(* CoDeSys 2.3 project: cy-wg-120-001.pro *)
(* Title: cy-wg-24 - ClevergyAS *)
(* Author: Andrea Laini *)
(* Libraries: mod_com.lib 16.5.13 14:00:50, SerComm.lib 16.5.13 14:00:50, Serial_Interface_01.lib 22.4.13 12:50:14, WagoLibLed.lib 17.6.13 10:40:56, Modb_l05.lib 13.5.15 10:30:08, Util.lib 16.5.13 14:00:50, SysLibFile.lib 16.5.13 14:00:50, SysLibRtc.lib 16.5.13 14:00:50, SysLibSockets.lib 22.5.14 16:16:32, SysLibEvent.lib 16.5.13 14:00:50, SysLibPlcCtrl.lib 16.5.13 14:00:50, Standard.lib 20.5.14 08:13:26, Iecsfc.lib 16.5.13 14:00:50, SYSLIBCALLBACK.LIB 16.5.13 14:00:50 *)

(* PLC configuration (modules and I/O channels)
0750-9999/0400-0004 4 DI Generic [Type_1_4_Channels] node 0, in %IB0 out %QB0
  VPN_ST2 AT %IX0.0 [BOOLOnX_I] I 1: Digital Input
  INT01 AT %IX0.1 [BOOLOnX_I] I 2: Digital Input
  KEY_QE_ST AT %IX0.2 [BOOLOnX_I] I 3: Digital Input
  INT02 AT %IX0.3 [BOOLOnX_I] I 4: Digital Input
Modbus variables [PFC200MODBUS] node 1, in %IB0 out %QB0 {PlcStopBehaviour = 1; FiledbusErrorBehaviour = 1; TcpOperation = 0; TcpPort = 502; TcpTimeout = 600; UdpOperation = 0; UdpPort = 502; RtuOperation = 0; NodeId = 200; ResponseTimeout = 5000; Interface = 0; Baud = 38400; StopBits = 2; Parity = 0; FlowCtrl = 0; PhysInterface = 1}
Modbus-Master [MB_MASTER] node 2, in %IB0 out %QB0
*)

(* Task configuration *)
TASK Main (PRIORITY := 6, INTERVAL := T#10ms);
	PLC_PRG();
END_TASK
TASK SystemCheck (PRIORITY := 14, INTERVAL := T#50ms);
	PLC_SYS_FAST();
END_TASK
TASK RTC (PRIORITY := 15, INTERVAL := T#500ms);
	RTC_Update();
END_TASK

(* Global variable list: Global_Constants *)
VAR_GLOBAL CONSTANT

	Plant_NAME			: STRING :='cySN:120 ITB CENE SOLARFAST cyVER:1';
	Plant_SN			: DWORD  :=120;		(* S/N Impianto di telecontrollo *)
	Plant_SW_VER		: WORD   :=1;		(* Versione SW installata *)

	Plant_INV			: BYTE	 :=2;
	Plant_STR			: BYTE	 :=6;

	(* Filesystem *)
	FilesPath  			: STRING :='/media/sd/';

	(* Colour Visu *)
	COLOR_RED			: DWORD := 16#2020F0;
	COLOR_YELLOW		: DWORD	:= 16#20F0F0;
	COLOR_GREEN			: DWORD	:= 16#20F020;

	(* TCP Logger *)
	Logger_SERVER		: STRING:='';
	Logger_IP			: STRING:='178.33.227.41';
	Logger_PORT			: WORD  :=80;
	Logger_GETSTART		: STRING:='GET /cygmsrv/SFgm.ashx?';
	Logger_GETEND		: STRING:='$R$N$R$N';
	Logger_CHECK		: STRING:='True';
	Logger_CRLF			: STRING:='$R$N';
	Logger_DataFile		: STRING:='/media/sd/LOG.DAT';
	Logger_DataFileOld	: STRING:='/media/sd/LOG.BCK';
	Logger_IndexFile	: STRING:='/media/sd/LOG.IDX';
	Logger_ConnRetries	: BYTE:=5;
	Logger_RecoverMsgs	: BYTE:=25;

	(* TCP Remote *)
	Remote_PORT			: WORD  :=10;
	Remote_WELCOME		: STRING:='Connected$R$N';
	Remote_OK			: STRING:='OK$R$N';
	Remote_ERROR		: STRING:='ERROR$R$N';

	(* TCP Sockets *)
	MAX_SEND_TCP_SERVER					 : DWORD:=3000;(*60000*)
	MAX_RECEIVE_TCP_SERVER				 : DWORD:=3000;
	MAX_RECEIVE_TCP_SERVER_SOCKET	 	 : DWORD:=1500;
	MAX_SEND_TCP_CLIENT					 : DWORD:=3000;(*15000*)
	MAX_RECEIVE_TCP_CLIENT				 : DWORD:=1500;
	MAX_RECEIVE_TCP_CLIENT_SOCKET		 : DWORD:=1500;
	MAX_RECEIVE_UDP_SERVER				 : INT  :=1472;
	MAX_RECEIVE_UDP_CLIENT				 : INT  :=1472;
	CONNECT_WATCHDOG_TIME				 : TIME :=t#10s;

END_VAR

(* Global variable list: Global_Retain *)
VAR_GLOBAL RETAIN PERSISTENT
	Mode_Manual : BOOL := FALSE;

	(* Offset correction in case of energy counter reset *)
	Offset		:	ARRAY [1..Plant_INV] OF DINT;

	(* Last value read (Stored in nvm to be sure that in case of a register reset after a voltage dropout, accumulated energy
       is not lost)	*)
	Old_Esup	:	ARRAY [1..Plant_INV] OF DINT;

END_VAR

(* Global variable list: Global_Variables *)
VAR_GLOBAL

	SYS    	: 	typ_SYS;
	Logger 	: 	typ_Logger;

	Lamp	:	LAMP_AL_GENERALE; (* Per gestione allarme generico impianto *)

	(**** PLANT OBJECTS ****)

	(* Define the handler for the ModBus communication	*)
	MODB01		:	obj_MODBUS := (ID:=1, COM:=0, BAUDRATE:=BAUD_38400, RS485:=TRUE);

	(* Define handlers for different objects in the plant; using array permits a better and immediate access *)
	INV			:	ARRAY[1..Plant_INV] OF obj_MODBUS_INV_SUNWAYTG;
	STR			:	ARRAY[1..Plant_STR] OF obj_MODBUS_STR_ES889;

	(**** SIMULATION ONLY ****)
	(*...*)
END_VAR

(* Data type in Logger *)
TYPE en_Logger_ErrLev :
(
	EL_Log			:=0,
	EL_Wrn			:=1,
	EL_Alarm		:=2,
	EL_AlarmStop	:=3,

	EL_Evt			:=4
);
END_TYPE

(* Data type in Logger *)
TYPE en_Logger_Status :
(
	S_Logger_UNKNOWN := 0,
	S_Logger_IDLE,
	S_Logger_WAITCONN,
	S_Logger_WAITTX,
	S_Logger_WAITRESP,
	S_Logger_ERROR
);
END_TYPE

(* Data type *)
TYPE en_SYS_Objects :
(
	EO_SYS		:=0,  (* PLC *)
	EO_VPN		:=1,  (* VPN *)
	EO_DOOR		:=2,  (* Door & access control *)

(*NEW*)EO_SWITCH	:= 3,

	EO_CAL		:=10, (* Caldaia *)
	EO_CIR		:=11, (* Circolatore *)
	EO_CRON		:=12, (* Crono-termostato *)
	EO_VRD		:=13, (* Valvola miscelatore pannelli *)
	EO_CTL		:=14, (* Contalitri *)
	EO_CTB		:=15, (* Contabilizzatore *)
	EO_TPV		:=16, (* Temperature probes values *)
	EO_PPV		:=17, (* Pressure probes values *)
	EO_PBV		:=18, (* Over-Pressure Alarms *)
	EO_TBV		:=19, (* Over-Temperature Alarms *)
	EO_PMV		:=20, (* Under-Pressure Alarms *)
	EO_GRU		:=21, (* Gruppo termico *)
	EO_PDC		:=22, (* Pompa di calore *)
	EO_SOL		:=23, (* Pannello solare termico *)
	EO_ESOL		:=24, (* Pannello solare fotovoltaico *)
	EO_GAS		:=25, (* Contatore GAS *)
	EO_PORT		:=26, (* Misuratore di portata *)
	EO_FPV		:=27, (* Flow probes values *)
	EO_ANZ		:=28, (* Analizzatore di rete *)
	EO_SCA		:=29, (* Signal Control Alarms *)
	EO_LUX		:=30, (* Illumination point *)
	EO_PSG		:=31, (* Sensore di passaggio *)

(*NEW*)EO_INV		:=36, (* Inverter *)
(*NEW*)EO_STR		:=37, (* Smart string box *)

	EO_ZGW			:=200,  (* ZigBee - Gateway *)
	EO_ZRM			:=201,	(* ZigBee - Repeater *)
	EO_ZREL			:=202,	(* ZigBee - Actuator rele *)
	EO_ZTHL			:=203,	(* ZigBee - Temperature Sensor *)

	EO_ASGW			:=250,	(* ASi - Gateway *)
	EO_ASCBI		:=251,	(* ASi - Input Board, Ciabatta *)

	EO_LON			:=1000, (* Bus - LON *)
	EO_MODBUS		:=1001, (* Bus - MODBUS *)
	EO_MBUS			:=1002, (* Bus - M-BUS *)
	EO_MODBUS_TCP	:=1003, (* Bus - MODBUS TCP *)

	EO_GENERIC		:=9000, (* Generic dataset *)
	EO_EXPO			:=9001 (* EXPO dataset *)
);
END_TYPE

(* Data type *)
TYPE en_SYS_Status :
(
	S_UNKNOWN  := 0,
	S_STARTUP,
	S_INIT_RTC,
	S_INIT_VAR,
	S_AUTOTEST,
	S_RUNNING,
	S_SHUTDOWN,
	S_HALT
);
END_TYPE

(* Data type in Logger *)
TYPE typ_Logger :
STRUCT
	Status		: en_Logger_Status;

	SendReq		: BOOL;
	SendIdx		: DWORD;
	SendData	: ARRAY [0..MAX_SEND_TCP_CLIENT] OF BYTE;
	SendLen		: DINT;

	TData		: ARRAY [0..MAX_SEND_TCP_CLIENT] OF BYTE;
	TLen		: DINT;

	LastIdxPos	: DWORD;

	(* Temporary variables used by objects *)
	s1			: STRING(256);
	i1			: WORD;

END_STRUCT
END_TYPE

(* Data type in Plant_Objects *)
TYPE typ_MODBUS_INV_SUNWAYTG : (* updated by Diego Bernini on 2016-02-18 *)
STRUCT
		(**** General measurements (see Programming manual) ****)
		Vpv_ref		:	WORD;	(* e-1 V*)
		f			:	INT;	(* e-2 Hz *)
		pf			:	WORD;	(* e-2 *)
		P			:	INT;	(* e-1 kW *)	(* Power supplied to the net b the inverter *)
		Pr			:	INT;	(* e-1 kVAr *)	(* Reactive power supplied to the net b the inverter *)
		Pa			:	INT;	(* e-1 kVA *)	(* Appearent power supplied to the net b the inverter *)
		Vinv		:	WORD;	(* e-1 V *)		(* Inverter output voltage, before output tf *)
		Vmain	 	:	WORD;	(* e-1 V *)		(* Main voltage, after output tf *)
		Iinv		:	WORD;	(* e-1 A *)		(* As voltage *)
		Imain		:	WORD;	(* e-1 A *)		(* AS voltage *)
		Vpv			:	WORD;	(* e-1 V *)		(* PV field voltage measured by the inverter *)
		Ipv			:	WORD;	(* e-1 A *)		(* PV current measured by the inverter *)
		Ppv			:	INT;	(* e-1 kW *)	(* Power generated by the PV *)

		(**** Energy ****)
		Esup_ExtCtr1:	DINT;	(* e-2 kWh *)	(* Global active energy supplied to the net *) (* updated *)
		ExtCtr2		:	DINT;	(* e-2 kWh *)
		Epv			:	DWORD;	(* e-2 kWh *)	(* Global produced energy since start *)

		(**** Temeprature ****)
		Tboard		:	INT;	(* e-1 °C *)	(* Control board temperature *)
		Tigbt		:	INT;	(* e-1 °C *)	(* Igbt temperature *)

		(**** Digital Input ****)
		ClampStatus	:	WORD;

		(**** Main measurements (otherwise not specified, all measurements are referred to the mains, therefore AFTER output tf ****)
		Vrms_rs		:	WORD;	(* e-1 V *)
		Vrms_st		:	WORD;
		Vrms_tr		:	WORD;
		Irms_r		:	INT;	(* e-1 A *)
		Irms_s		:	INT;
		Irms_t		:	INT;
		PLLStatus	:	WORD;
		MainStatus2	:	WORD;
		MainStatus1	:	WORD;
		Iinv_rms_r	:	INT;	(* e-1 A *)		(* Measured between inverter and tf *)
		Iinv_rms_s	:	INT;
		Iinv_rms_t	:	INT;
		Iimbalance	:	WORD;	(* e-1 *)
		Vrms_r		:	WORD;	(* e-1 V *)
		Vrms_s		:	WORD;
		Vrms_t		:	WORD;
		P_r			:	INT;	(* e-1 kW *)
		P_s			:	INT;
		P_t			:	INT;
		Pr_r		:	INT;	(* e-1 kW *)
		Pr_s		:	INT;
		Pr_t		:	INT;

		(**** Inverter Status (see Programming manual) ****)
		Status		:	WORD;
		ActiveAlarm	:	WORD;
		Insulation	:	WORD;
		Event		:	WORD;
		OpTime		:	DWORD;	(* e-0.7 s *)
		SuppTime	:	DWORD;	(* e-0.7 s *)

END_STRUCT
END_TYPE

(* Data type in Plant_Objects *)
TYPE typ_MODBUS_INV_SUNWAYTG_His :
STRUCT
		AlarmID		:	WORD;
		SuppTime	: 	DWORD;
		OpTime		:	DWORD;
		InvStatus	:	WORD;
		Vpv_ref		:	WORD;
		Vpv			:	WORD;
		Vmain		:	WORD;
		Status2		:	WORD;
		Status1		:	WORD;
		Tboard		:	INT;
		Tigbt		:	INT;
		I_u			:	INT;
		I_v			:	INT;
		I_w			:	INT;
		ClampStatus	:	WORD;
		DigOutput	:	WORD;
		IgbtFault	:	WORD;
		Psupp		:	DWORD;
		Epv			:	DWORD;

END_STRUCT
END_TYPE

(* Data type in Plant_Objects *)
TYPE typ_MODBUS_STR_ES889 :
STRUCT

	(* GENERAL MEASUREMENTS *)
	(* String current *)
	Istring1	:	WORD;			(* e-2 A *)
	Istring2	:	WORD;
	Istring3	:	WORD;
	Istring4	:	WORD;
	Istring5	:	WORD;
	Istring6	:	WORD;
	Istring7	:	WORD;
	Istring8	:	WORD;
	Iavg		:	WORD;
	Imax		:	WORD;
	Imin		:	WORD;

	(* Optional sensors *)
	Radiation_h	:	WORD;			(* e-1 W/m2	,	Radiation on the horizontal plane *)
	Radiation_m	:	WORD;			(*			,	Radiation on modules plane *)
	Tmodule		:	INT;			(* e-1 °C	,	Module temperature *)
	Tenv		:	INT;			(*			,	Environment temperature *)
	Vwind		:	WORD;			(* e-1 m/s	,	Wind speed *)
	Tboard		:	INT;			(* e-1 °C	,	Board temperature *)

	(* FUNCTIONING STATUS *)
	M018		:	WORD;
	M019		:	WORD;
	M020		:	WORD;

	(* TIMING *)
	SuppTime	:	DWORD;			(* s ???? *)
	OpTime		:	DWORD;			(* s ???? *)

	(* String mask	*)
	Mask		:	WORD;

	(* Panels number	*)
	Panels		:	WORD;

END_STRUCT
END_TYPE

(* Data type in Plant_Objects *)
TYPE typ_MODBUS_STR_ES889_His :
STRUCT

	M018		:	WORD;
	M020		:	WORD;
	Tmodule		:	INT;			(* e-1 °C	,	Module temperature *)
	SuppTime	:	DWORD;
	OpTime		:	DWORD;

END_STRUCT
END_TYPE

(* Data type in Plant_Objects *)
TYPE typ_MODBUS_VAR : (* Gestione parametri MODBUS *)
STRUCT
	SlaveAddress	: BYTE;
	FunCode			: BYTE;
	FunAddress		: WORD;
	Refresh_Time	: BYTE; (* 0:No refresh x:Refresh in seconds *)
	Refresh_Cnt		: BYTE; (* INTERNAL *)
	Variable		: POINTER TO ARRAY [0..124] OF WORD;	(* For classical ModBus it has to be equal to "typModbusResponse.Data"
																that is an array of 125 word ([0..124]) *)
	Variable_Size	: BYTE;
	Variable_Mirror : WORD; (* INTERNAL [Force refresh on read variables when <>0] *)
END_STRUCT
END_TYPE

(* Data type *)
TYPE typ_SYS :
STRUCT
	Status			: en_SYS_Status;
	Warning			: BOOL;
	Alarm			: BOOL;
	AlarmStop		: BOOL;

	Time_LogString	: STRING;
	Time_Year		: WORD;
	Time_Month		: BYTE;
	Time_Day		: BYTE;

	Time_CT_DT		: DT;
	Time_CT_Day		: WORD;
	Time_CT_Quarter	: BYTE;

	LastLogs_Idx	: BYTE;
	LastLogs_Dat	: ARRAY[0..5] OF STRING;
	LastLogs_Msg	: ARRAY[0..5] OF STRING;

END_STRUCT
END_TYPE

(* Data type in Plant_Objects *)
TYPE typ_VisuStrutturaMbus :
STRUCT

	sdNodoPresente: STRING(16);
	sdEnergia: STRING(16);
	sdPotenza: STRING(16);
	sdVolume: STRING(16);
	sdFlow: STRING(16);
	sdTempIngresso: STRING(8);
	sdTempaUscita: STRING(8);
	sdTempDelta: STRING(8);

END_STRUCT
END_TYPE

(* POU PLC_PRG, ST *)
PROGRAM PLC_PRG
VAR
	Timer1: TON; (* Logger timer *)

	i	  : BYTE;
	status : BYTE;
END_VAR
(******************************************************************************
 ****        		MAIN TASK CODE  (called every 10ms)                    ****
 ******************************************************************************

	Network setup:
		IP  = 192.168.100.2 | MSK = 255.255.255.0
		GW	= 192.168.100.1 | DNS = 192.168.100.1
		SNTP = 193.204.114.232 (3600s) ==> 192.168.100.3

*)

(*==============================*)
(*===== Main status machine ====*)
(*==============================*)
Main_Stm();

(*==============================*)
(*== Running cycle operations ==*)
(*==============================*)
IF SYS.Status>S_INIT_VAR THEN
	(* Execute cycle processes *)
	MODB01();

	FOR i:=1 TO Plant_INV BY 1 DO INV[i](ModBus:=MODB01, retryErrMax:=1);	END_FOR

	FOR i:=1 TO Plant_STR BY 1 DO STR[i](ModBus:=MODB01, retryErrMax:=1);   END_FOR

END_IF

(*==============================*)
(*== System cycle operations ===*)
(*==============================*)
(* Execute TCP processes *)
Logger_Proc();
Remote_Proc();
(* Update user led *)
(*USRLED_Update();*)
(* Execute Cron Editor commands *)
(*
CronEd();
*)
(* External resources *)
(*

*)

(**** SIMULATION ONLY ****)
(*...*)
END_PROGRAM
ACTION Main_Stm:
CASE Sys.Status OF

	S_STARTUP:
		Sys.Status:=S_INIT_RTC;

	S_INIT_RTC:
		(* Check RTC and update from network *)
		RTC_Update();
		(* Check time *)
		IF Sys.Time_Year>2000 THEN
			Sys.Status:=S_INIT_VAR;
		END_IF

	S_INIT_VAR:
		OBJ_Definition();

		LogEv(EL_Wrn,EO_SYS,0,1,CONCAT('System_startup_v',WORD_TO_STRING(Plant_SW_VER)));
		Sys.Status:=S_RUNNING;

	S_RUNNING:

		status :=0;
		FOR i:=1 TO Plant_INV BY 1 DO IF INV[i].Status_Log=1 THEN status :=1;  END_IF	END_FOR

		FOR i:=1 TO Plant_STR BY 1 DO IF str[i].Status_Log=1 THEN status :=1; END_IF END_FOR

		FOR i:=1 TO Plant_INV BY 1 DO IF INV[i].Status_Log=2 THEN status :=2;  END_IF	END_FOR

		FOR i:=1 TO Plant_STR BY 1 DO IF str[i].Status_Log=2 THEN status :=2; END_IF END_FOR

		Lamp( Allarme:=	(status=2),
			  Warning:=  (status=1),
			  SistemaInAllarme => Sys.Alarm,
			 SistemaWarning => Sys.Warning
			 );

		Timer1(IN:=NOT Timer1.Q,PT:=T#5m);
		IF Timer1.Q THEN
			(* Trig logger *)
			LogTrig();
			(* Execute temporary CSV logger *)
			(*CSV_Log();*)
		END_IF

	S_SHUTDOWN:
		(* Stop sistema *)
		Sys.Status:=S_STARTUP;

	S_HALT:
		(* Aspetta uscita manuale *)
		Sys.Status:=S_STARTUP;

ELSE
	Sys.Status:=S_STARTUP;
END_CASE;
END_ACTION
ACTION OBJ_Definition:
(**** Define Plant Objects ****)

(* Inverter *)
INV[1].ID := 1;		INV[1].Address := 2;
INV[2].ID := 2;		INV[2].Address := 3;


(* StringBox *)
STR[1].ID := 1;		    STR[1].Address :=10;
STR[2].ID := 2;		    STR[2].Address := 11;
STR[3].ID := 3;		    STR[3].Address := 12;
STR[4].ID := 4;		    STR[4].Address := 13;
STR[5].ID := 5;		    STR[5].Address := 14;
STR[6].ID := 6;		    STR[6].Address := 15;
END_ACTION

(* POU TCP_Logger/Logger_Proc, ST *)
PROGRAM Logger_Proc
VAR
	c1:         	TCPCLIENT;

	Open:	    	BOOL;
	IpAddr:			DWORD;
	InetAddr:		DWORD;
	Connected:  	BOOL;
	Error:      	DINT;
	TxTrig:     	BOOL;
	RxData:			ARRAY [0..MAX_RECEIVE_TCP_CLIENT] OF BYTE;
	RxLen:			DINT;

	Retry:			BYTE;	(* Counter for connection retries *)
	Recovered:		BYTE;	(* Counter for recovered unsent messages *)

	i:				DINT;
	pos:			DWORD;
	hFile:			DWORD;

END_VAR
(*=== State machine ===*)
CASE Logger.Status OF

	S_Logger_UNKNOWN:
		(* Startup *)
		Logger.SendReq:=FALSE;
		Open:=FALSE;
		Logger.Status:=S_Logger_IDLE;

	S_Logger_IDLE:
		(* Wait request *)
		IF Logger.SendReq THEN
			(* Resolve server name or use static IP *)
			IF LEN(Logger_SERVER)=0 THEN
				InetAddr:=SysSockInetAddr(Logger_IP);
			ELSE
				IpAddr:=SysSockGetHostByName(ADR(Logger_SERVER));	(* Get the IP address by the DNS *)
				DWORDSWAP(pIn:=ADR(IpAddr), pOut:=ADR(InetAddr));
			END_IF
			TxTrig:=FALSE;
			RxLen:=0;
			(* Open connection *)
			Open:=TRUE;
			Logger.Status:=S_Logger_WAITCONN;
		END_IF

	S_Logger_WAITCONN:
		(* Wait connection *)
		IF Connected THEN
			(* Send data *)
			TxTrig:=TRUE;
			Logger.Status:=S_Logger_WAITTX;
		END_IF
		IF Error>0 THEN
			Open:=FALSE;
			Logger.Status:=S_Logger_ERROR;
		END_IF

	S_Logger_WAITTX:
		(* Wait transmission *)
		IF NOT TxTrig THEN
			Logger.Status:=S_Logger_WAITRESP;
		END_IF
		IF Error>0 THEN
			Open:=FALSE;
			Logger.Status:=S_Logger_ERROR;
		END_IF

	S_Logger_WAITRESP:
		(* Wait response *)
		IF Connected=FALSE (* OR TIMEOUT!! *) THEN
			Open:=FALSE;
			(* Check response *)
			IF RxLen>=4 AND CHKSTRING(pString:=ADR(RxData), pPattern:=ADR(Logger_CHECK)) THEN
			(* If "RxLen" is of the right size and function "CHKSTRING" has not return "FALSE"	*)
				Logger.SendReq:=FALSE;
				Retry:=0;
				(* Check unsent messages to flush *)
				IF Recovered<Logger_RecoverMsgs THEN
					MsgChk();
					IF Logger.SendReq=TRUE THEN
						Recovered:=Recovered+1;
					ELSE
						Recovered:=0;
					END_IF
				ELSE
					Recovered:=0;
				END_IF
				Logger.Status:=S_Logger_IDLE;
			ELSE
				Logger.Status:=S_Logger_ERROR;
			END_IF
		END_IF

	S_Logger_ERROR:
		(* Connection error or send failure *)
		Retry:=Retry+1;
		IF Retry>Logger_ConnRetries THEN
			(* Save message as unsent *)
			MsgSave();
			Logger.SendReq:=FALSE;
			Retry:=0;
		END_IF
		Logger.Status:=S_Logger_IDLE;

ELSE
	Logger.Status:=S_Logger_UNKNOWN;
END_CASE


(*=== Execute client lib ===*)
c1(
	xOpenConnection			:= Open,
	dwInetAddr 				:= InetAddr,
	wPortNumber				:= Logger_PORT,
	ptSendData				:= ADR(Logger.SendData),
	diSendCount				:= Logger.SendLen,
	tConnectWatchdogTime	:= t#10s,
	xStartSend				:= TxTrig,
	aReceiveBuffer			:= RxData,
	diReceiveCount			:= RxLen,
	xConnected				=> Connected,
	diError					=> Error
);

(*=== Process Rx data ===*)
(*IF RxLen>0 THEN
	RxLen:=0;
END_IF*)
END_PROGRAM
ACTION MsgChk:
(* Open index file *)
hFile:=SysFileOpen(Logger_IndexFile,'r');
IF hFile=0 THEN
	(* File doesn't exist, no pending message *)
	RETURN;
END_IF
(* Search oldest message to recover *)
SysFileSetPos(hFile,Logger.LastIdxPos);		(* Set the pointer to last position *)
Logger.SendLen:=0;
REPEAT
	SysFileRead(hFile, ADR(Logger.SendIdx), SIZEOF(Logger.SendIdx));
	pos:=SysFileGetPos(hFile);
	SysFileRead(hFile, ADR(Logger.SendLen), SIZEOF(Logger.SendLen));
UNTIL
	SysFileEOF(hFile) OR Logger.SendLen<>0		(* If equal to 0 means data not stored or deleted *)
END_REPEAT
SysFileClose(hFile);
(* Delete index file when all messages are recovered *)
IF Logger.SendLen=0 THEN
	Logger.LastIdxPos:=0;
	SysFileDelete(Logger_IndexFile);
	RETURN;
END_IF
(* Recover message data *)
hFile:=SysFileOpen(Logger_DataFile,'r');
IF hFile<>0 THEN
	SysFileSetPos(hFile,Logger.SendIdx);
	SysFileRead(hFile,ADR(Logger.SendData),Logger.SendLen);
	Logger.SendReq:=TRUE;									(* Re-trigger another transmission *)
	SysFileClose(hFile);
END_IF
(* Clear index entry *)
hFile:=SysFileOpen(Logger_IndexFile,'a');
IF hFile<>0 THEN
	SysFileSetPos(hFile,pos);
	i:=0;
	SysFileWrite(hFile, ADR(i), 4);			(* Since the size is in number of byte, that clears only the Idx, not the Len *)
	Logger.LastIdxPos:=SysFileGetPos(hFile);
	SysFileClose(hFile);
END_IF
END_ACTION
ACTION MsgSave:
(* Add log position in recovery indexes *)
hFile:=SysFileOpen(Logger_IndexFile,'a');
SysFileWrite(hFile, ADR(Logger.SendIdx), SIZEOF(Logger.SendIdx));
SysFileWrite(hFile, ADR(Logger.SendLen), SIZEOF(Logger.SendLen));
SysFileClose(hFile);
END_ACTION

(* POU Utils Functions/TCPCLIENT, ST *)
FUNCTION_BLOCK TCPCLIENT
(***********************************************************************************************************	*)
(* Version: 1.3b                        			          													*)
(* Date: 28.10.2014                   				          							            			*)
(***********************************************************************************************************	*)
(* WAGO Kontakttechnik GmbH Hansastr. 27 32423 Minden(Westf.)													*)
(* Tel. +0049 571/887-0 Fax. +0049 571/887-0																	*)
(* Author: VB																									*)
(***********************************************************************************************************	*)
(*Description:	A TCP client to read and write data with additional connection watchdog							*)
(*History:																										*)
(*Version 1.3b: 28.10.2014: Use DWORD address for IP (Andrea Ravasio)											*)
(*Version 1.3: 11.02.2011: Changes according to 750-880/881											 			*)
(*Version 1.2: 29.08.2007 Bugfix TCP Client																		*)
(*Version 1.1: 15.01.2007 Changes according to FW11																*)
(*Version 1.0: 09.03.2006 Release																				*)
(***********************************************************************************************************	*)
VAR CONSTANT
	STATE_CREATE     				 : BYTE:= 0;
	STATE_OPEN     					 : BYTE:= 1;
	STATE_IOCTL    					 : BYTE:= 2;
	STATE_CONNECT     				 : BYTE:= 10;
	STATE_TX       					 : BYTE:= 20;
	STATE_RX       					 : BYTE:= 30;
	STATE_CLOSE    					 : BYTE:= 40;
	STATE_ERROR_TRAP			     : BYTE:= 200;
END_VAR

VAR_INPUT
	xOpenConnection					: BOOL;
	dwInetAddr						: DWORD; (* <== Use SysSockInetAddr() value or
													swapped bytes order of SysSockGetHostByName() value *)
	wPortNumber						: WORD;
	ptSendData						: POINTER TO ARRAY[0..MAX_SEND_TCP_CLIENT] OF BYTE;
	diSendCount						: DINT;
	tConnectWatchdogTime		    : TIME := t#10s;
END_VAR
VAR_OUTPUT
	xConnected						: BOOL;
	diError 						: DINT := 0;
END_VAR
(* ErrorCodes -----------------------------------------
	16#8001 => No socket descriptor available 
	16#8002 => SysSockSend returns -1 
	16#8003 => Socket was "gracefully closed" 
	16#8004 => switching to none blocking mode fails
	16#8005 => SysSockClose() returns FALSE 
    16#8006 => SysSockConnect() fails
    16#8007 => SysSockSend() fails
	16#8008 => error state machine 
	16#8009 => timeout while waiting for data from server 
------------------------------------------------------------*)
VAR_IN_OUT
	xStartSend							: BOOL;
	aReceiveBuffer						: ARRAY [0..MAX_RECEIVE_TCP_CLIENT] OF BYTE;
	diReceiveCount						: DINT;
END_VAR
VAR
	m_State								: BYTE := 0;
	m_ReceiveBuffer						: ARRAY [0..MAX_RECEIVE_TCP_CLIENT_SOCKET] OF BYTE;
	m_Socket							: DINT;
	m_AddressInfo						: SOCKADDRESS;
	m_BytesReceived						: DINT;
	m_diReturn							: DINT;
	m_xReturn							: BOOL;
	m_IoCtlParameter  					: DINT := 1; (* IOCTL-Parameter for non-blocking mode of sockets *)
	i									: INT;
	T_Connect							: TON;
	m_count								: DINT;
	diOption							: DINT := 1;
	m_Blocking   						: DINT := 0;
END_VAR
IF xOpenConnection THEN
	(* State maschine *)
	CASE  m_State OF

	(* -------------------------------------------------------------------------*)
	STATE_CREATE:
			(* create socket descriptor*)
			m_Socket := SysSockCreate(diAddressFamily	:= SOCKET_AF_INET,
													 diType		:= SOCKET_STREAM,
													 diProtocol := SOCKET_IPPROTO_TCP);
			IF m_Socket >= 0 THEN
			(*Set Push-Bit*)
				IF ADR(%MW0)=16#30000000  OR ADR(%MW0)=16#20000000 THEN (*841 or 881*)
					SysSockSetOption(
						diSocket:=m_Socket,
						diLevel:=6,
						diOption:=SOCKET_TCP_NODELAY,
						pOptionValue:=ADR(diOption),
						diOptionLength:=SIZEOF(diOption));
				ELSE
						;
				END_IF
				m_State := STATE_IOCTL; (* succesful *)
			ELSE
				diError := 16#8001;  (* no socket descriptor available *)
				m_State := STATE_ERROR_TRAP;
			END_IF

	(* -------------------------------------------------------------------------*)
	STATE_IOCTL: (* change  socket mode  to none blocking *)
		m_diReturn := SysSockIoctl( m_Socket, SOCKET_FIONBIO, ADR(m_IoCtlParameter));
		IF m_diReturn <> 0 THEN
			m_AddressInfo.sin_family := SOCKET_AF_INET;
			m_AddressInfo.sin_port := SysSockNtohs(wPortNumber);
			m_AddressInfo.sin_addr := dwInetAddr;
			m_State := STATE_CONNECT;
		ELSE
			diError := 16#8004;  (* switching to none blocking mode fails *)
			m_State := STATE_ERROR_TRAP;
		END_IF


	(* -------------------------------------------------------------------------*)
	STATE_CONNECT: (* connect with server *)
		T_Connect(IN:=TRUE , PT:=tConnectWatchdogTime);(*activate watchdog for establishing connection to a server*)
		m_xReturn := SysSockConnect ( m_Socket, ADR(m_AddressInfo),  SIZEOF(m_AddressInfo));
		IF m_xReturn THEN (* succesful *)
			IF xStartSend THEN
				m_State := STATE_TX;(*transmit data*)
			ELSE
				m_State := STATE_RX;(*wait for data from server*)
			END_IF
			xConnected:=TRUE;
			T_Connect(IN:=FALSE);
		ELSE
			IF T_Connect.Q THEN
				diError := 16#8006;  (* connect fails *)
				xConnected:=FALSE;
				T_Connect(IN:=FALSE);
				m_State := STATE_ERROR_TRAP;
				SysSockClose( m_Socket);
			ELSE
				m_State := STATE_CONNECT;(*client still  tries to set up connection*)
			END_IF
		END_IF


	STATE_TX:	 (* send TCP-message *)
		m_diReturn := SysSockSend(diSocket := m_Socket,
								  pbyBuffer := ADR(ptSendData^[0]),
								  diBufferSize := diSendCount-m_count,
								  diFlags := 0);

		CASE m_diReturn OF
		-1:	(* ERROR *)
			T_Connect(IN:=TRUE , PT:=CONNECT_WATCHDOG_TIME);(*activate watchdog to check communication*)
			IF t_Connect.Q THEN
				diError := 16#8007;
				T_Connect(IN:=FALSE);
				m_State:=STATE_CLOSE;
			END_IF
		0: (* socket was "gracefully closed" *)
			m_State := STATE_CLOSE;
			diError := 16#8003;
		ELSE (* succesful *)
			m_count:=m_count+m_diReturn;
			IF m_count>=diSendCount THEN
				diError := 16#0000;
				m_State := STATE_RX;
				m_count:=0;
				xStartSend:=FALSE;
			END_IF
			T_Connect(IN:=FALSE);
		END_CASE

	(* -------------------------------------------------------------------------*)
	STATE_RX: (* process receive data *)
			m_BytesReceived := SysSockRecv(	diSocket 	:= m_Socket,
										pbyBuffer 	:= ADR(m_ReceiveBuffer),		(* Address of receive buffer *)
										diBufferSize:= SIZEOF(m_ReceiveBuffer),
										diFlags		:= 0);

			CASE m_BytesReceived OF
			-1:	(* No data available or error occured *)
				T_Connect(IN:=TRUE , PT:=tConnectWatchdogTime);(*activate watchdog to check communication*)
				IF t_Connect.Q THEN
					diError:=16#8009;
					T_Connect(IN:=FALSE);
					m_State:=STATE_CLOSE;
				END_IF
				IF xStartSend THEN
					m_State:=STATE_TX	;(* WAIT IN THIS STATE  and check for arriving data or new send command*)
				END_IF;
			0: (* socket was "gracefully closed"  *)
				m_State:=STATE_CLOSE;
				diError := 16#8003;
			ELSE (* succesful *)
				diError := 16#0000;
				T_Connect(IN:=FALSE);
				(* Copy received data into receive buffer *)
				FOR i:= 0 TO DINT_TO_INT(m_BytesReceived	)-1 DO
					aReceiveBuffer[diReceiveCount]:= m_ReceiveBuffer[i];
					diReceiveCount:=(diReceiveCount+1) MOD SIZEOF(aReceiveBuffer);
				END_FOR

			END_CASE

	(* -------------------------------------------------------------------------*)
	STATE_CLOSE : (* close socket *)
		IF ADR(%MW0)=16#30000000  OR ADR(%MW0)=16#20000000 THEN (*841 or 881*)
			;
		ELSE
			SysSockShutdown(m_Socket, 0);;(*870*)
		END_IF
		m_xReturn := SysSockClose( m_Socket);
		m_Socket := -1;
		m_State := 0; (* succesful *)
		xConnected:=FALSE;
		T_Connect(IN:=FALSE);
	(* -------------------------------------------------------------------------*)
	STATE_ERROR_TRAP: (* error handling *)
		xConnected:=FALSE;

	ELSE  (* Bad FSM code trap  *)
			m_State:= STATE_ERROR_TRAP;
			diError:= 16#8008;
	END_CASE

ELSE(*close connection*)
	IF m_Socket >= 0 THEN
		IF ADR(%MW0)=16#30000000  OR ADR(%MW0)=16#20000000 THEN (*841 or 881*)
			;
		ELSE
			SysSockShutdown(m_Socket, 0);;(*870*)
		END_IF
		SysSockClose( m_Socket);
	END_IF
	m_Socket := -1;
	diError := 16#0000;
	m_State := STATE_CREATE;
	xConnected:=FALSE;
	T_Connect(IN:=FALSE);
END_IF
END_FUNCTION_BLOCK

(* POU Utils Functions/DWORDSWAP, ST *)
FUNCTION DWORDSWAP:BOOL
VAR_INPUT
	pIn:POINTER TO ARRAY[1..4] OF BYTE;
	pOut:POINTER TO ARRAY[1..4] OF BYTE;
END_VAR
VAR
END_VAR
pOut^[1]:=pIn^[4];
pOut^[2]:=pIn^[3];
pOut^[3]:=pIn^[2];
pOut^[4]:=pIn^[1];
END_FUNCTION

(* POU Utils Functions/CHKSTRING, ST *)
FUNCTION CHKSTRING : BOOL
VAR_INPUT
	pString: POINTER TO BYTE;
	pPattern: POINTER TO BYTE;
END_VAR
VAR
END_VAR
CHKSTRING:=TRUE;
WHILE pPattern^<>0 AND CHKSTRING DO
	IF pPattern^<>pString^ THEN CHKSTRING:=FALSE; END_IF
	pString:=pString+1;
	pPattern:=pPattern+1;
END_WHILE
END_FUNCTION

(* POU TCP_Remote/Remote_Proc, ST *)
PROGRAM Remote_Proc
VAR
	s1:         	TCPSERVER;
	Enable: 		BOOL;
	Connected: 		BOOL;
	Error: 			DINT;

	TxData:			ARRAY [0..MAX_SEND_TCP_SERVER] OF BYTE;
	TxLen:			DINT;
	TxTrig:			BOOL;

	RxData:			ARRAY [0..MAX_RECEIVE_TCP_SERVER] OF BYTE;
	RxLen:			DINT;

	Status:			DINT;

	(* Command interpreter *)

	Cmd_Buf:		ARRAY [0..MAX_RECEIVE_TCP_SERVER] OF BYTE;
	Cmd_Buf_U16:	POINTER TO WORD;
	Cmd_Buf_INT:	POINTER TO INT;
	Cmd_BufLen:		WORD;
	Cmd_St:			WORD;

	Cmd_Obj:		WORD;
	Cmd_ObjIdx:		WORD;
	Cmd_C:			WORD;
	Cmd_R:			WORD;
	Cmd_CLen:		WORD;
	Cmd_RLen:		WORD;

	i : WORD;
	j : INT;
	s2 : STRING;

	(* per aggiornare la data e l'ora *)
	SetAnno: INT;
	SetMese: INT;
	SetGiorno: INT;
	SetOra: INT;
	SetMinuti: INT;
	SetSecondi: INT;

	Plant_SW_VER: BOOL;
END_VAR
(*=== State machine ===*)
CASE Status OF
	0: (* Startup *)
		TxLen:=0; TxTrig:=FALSE;
		RxLen:=0;
		Enable:=TRUE;
		Status:=1;

	1: (* Wait incoming connection *)
		IF Connected THEN
			(* Log access *)(*
			LogEv(EL_Log,EO_VPN,1,5,'Remote');*)
			(* Send welcome message *)(*
			ADDSTRING(pTxData:=ADR(TxData), pString:=ADR(Remote_WELCOME), TxLen:=TxLen);
			TxTrig:=TRUE;*)
			(* Reset vars *)
			Cmd_BufLen:=0;
			Cmd_St:=0;
			Status:=2;
		END_IF
		IF Error>1 THEN
			Enable:=FALSE;
			Status:=0;
		END_IF

	2: (* Wait command *)
		IF RxLen>0 THEN
			(*=== Interpreter start ===*)
			IF Cmd_BufLen+(RxLen/2)>=MAX_RECEIVE_TCP_SERVER THEN
				(* ERROR *)
				Cmd_BufLen:=0;
			ELSE
				i:=HEXTORAW(pString:=ADR(RxData), StringLen:=DINT_TO_WORD(RxLen), pData:=ADR(Cmd_Buf[Cmd_BufLen]));
				Cmd_BufLen:=Cmd_BufLen+i;
			END_IF
			IF Cmd_BufLen>=8 THEN
				Cmd_Buf_U16:=ADR(Cmd_Buf[6]);
				IF Cmd_BufLen>=(8+Cmd_Buf_U16^) THEN	(* Right number of bytes has been received (8 of protocol + data) *)
					Cmd_CLen:=Cmd_Buf_U16^;
					Cmd_Buf_U16:=ADR(Cmd_Buf[0]); Cmd_Obj:=Cmd_Buf_U16^;
					Cmd_Buf_U16:=ADR(Cmd_Buf[2]); Cmd_ObjIdx:=Cmd_Buf_U16^;
					Cmd_Buf_U16:=ADR(Cmd_Buf[4]); Cmd_C:=Cmd_Buf_U16^;
					(* Log command *)(*
					s2:='RCmd_';		s2:=CONCAT(s2,WORD_TO_STRING(Cmd_Obj));
					s2:=CONCAT(s2,'_'); s2:=CONCAT(s2,WORD_TO_STRING(Cmd_ObjIdx));
					s2:=CONCAT(s2,'_'); s2:=CONCAT(s2,WORD_TO_STRING(Cmd_C));
					s2:=CONCAT(s2,'_');	s2:=CONCAT(s2,WORD_TO_STRING(Cmd_CLen));
					LogEv(EL_Log,EO_VPN,1,6,s2);*)
					(* Execute command *)
					Command();
					Cmd_BufLen:=0;
				END_IF
			END_IF
			(*=== Interpreter end ===*)
			RxLen:=0;
		END_IF
		IF NOT Connected THEN
			Status:=0;
		END_IF

ELSE
	Status:=0;
END_CASE


(*=== Execute server lib ===*)
s1(
	xEnable				:= Enable,
	wPortNumber			:= Remote_PORT,
	tServerTimeOut		:= t#15m,
	ptSendData			:= ADR(TxData),
	diSendCount			:= TxLen,
	xStartSend			:= TxTrig,
	aReceiveBuffer		:= RxData,
	diReceiveCount		:= RxLen,
	xClientConnected	=> Connected,
	diError				=> Error
);
END_PROGRAM
ACTION Cmd_CRON:
(* Check index *)(*
IF Cmd_ObjIdx<1 OR Cmd_ObjIdx>6 THEN
	Cmd_R:=2;
	RETURN;
END_IF

(* Process command *)
CASE Cmd_C OF

	1: (* GET PROFILE *)
		IF Cmd_CLen<>3 THEN
			Cmd_R:=4;
		ELSE
			(* Load profile *)
			CronEd.CN_Sel:=WORD_TO_BYTE(Cmd_ObjIdx);
			Cmd_Buf_U16:=ADR(Cmd_Buf[8]);
			CronEd.CN_YSel:=Cmd_Buf_U16^;
			CronEd.PR_Sel:=Cmd_Buf[10];
			CronEd.PR_Load_Exe();
			(* Copy data *)
			Cmd_RLen:=192;
			TxLen:=TxLen+RAWTOHEX(ADR(CronEd.PR.Setpoint),192,ADR(TxData[TxLen]));
		END_IF

	2: (* SET PROFILE *)
		IF Cmd_CLen<>(3+192) THEN
			Cmd_R:=4;
		ELSE
			(* Save profile *)
			CronEd.CN_Sel:=WORD_TO_BYTE(Cmd_ObjIdx);
			Cmd_Buf_U16:=ADR(Cmd_Buf[8]);
			CronEd.CN_YSel:=Cmd_Buf_U16^;
			CronEd.PR_Sel:=Cmd_Buf[10];
			MEMCPY(ADR(Cmd_Buf[11]),ADR(CronEd.PR.Setpoint),192);
			CronEd.PR_Save_Exe();
		END_IF

	5: (* GET CALENDAR MONTH *)
		IF Cmd_CLen<>3 THEN
			Cmd_R:=4;
		ELSE
			(* Load calendar *)
			CronEd.CN_Sel:=WORD_TO_BYTE(Cmd_ObjIdx);
			Cmd_Buf_U16:=ADR(Cmd_Buf[8]);
			CronEd.CN_YSel:=Cmd_Buf_U16^;
			CronEd.CA_Sel:=Cmd_Buf[10];
			CronEd.CA_Load_Exe();
			(* Copy data *)
			Cmd_RLen:=32;
			TxLen:=TxLen+RAWTOHEX(ADR(CronEd.CA.Profile),32,ADR(TxData[TxLen]));
		END_IF

	6: (* SET CALENDAR MONTH *)
		IF Cmd_CLen<>(3+32) THEN
			Cmd_R:=4;
		ELSE
			(* Save calendar *)
			CronEd.CN_Sel:=WORD_TO_BYTE(Cmd_ObjIdx);
			Cmd_Buf_U16:=ADR(Cmd_Buf[8]);
			CronEd.CN_YSel:=Cmd_Buf_U16^;
			CronEd.CA_Sel:=Cmd_Buf[10];
			MEMCPY(ADR(Cmd_Buf[11]),ADR(CronEd.CA.Profile),32);
			CronEd.CA_Save_Exe();
		END_IF

	9: (* CRON RESTART *)
		CASE Cmd_ObjIdx OF
			1: CRON01.InitOK:=FALSE;
			2: CRON02.InitOK:=FALSE;
			3: CRON03.InitOK:=FALSE;
			4: CRON04.InitOK:=FALSE;
			5: CRON05.InitOK:=FALSE;
			6: CRON06.InitOK:=FALSE;
		END_CASE

ELSE
	Cmd_R:=3;
END_CASE
*);
END_ACTION
ACTION Cmd_INV:
(* Check if object index out of range *)
IF Cmd_ObjIdx=0 OR Cmd_ObjIdx>Plant_INV THEN
	Cmd_R:=2;
	RETURN;
END_IF

(* Execute the command *)
CASE Cmd_C OF

	0,1,2,3,4,5,6,7:	(* Read ALARM FAULT LIST -> Choosen alarm of last 8 alarms with significant measurements will be returned		*)
		INV[Cmd_ObjIdx].FaultAddr := 7712 + Cmd_C * 32;		(* Set right address ModBus of first alarm to be read	*)


	8,9,10,11,12,13,14,15,16,17,18,19,20,21,22,23:	(* Read EVENTS FAULT LIST -> Choosen event of last 16 events will be sent	*)
		INV[Cmd_ObjIdx].FaultAddr := 5044 + (Cmd_C-8)*32;

ELSE
	Cmd_R:=3;
END_CASE

(* If response OK add requested data	*)
IF Cmd_R=0 THEN

	Cmd_RLen := 46;

	TxLen := RAWTOHEX(ADR(INV[Cmd_ObjIdx].FaultData.AlarmID),2,ADR(TxData[TxLen]));
	TxLen := RAWTOHEX(ADR(INV[Cmd_ObjIdx].FaultData.SuppTime),4,ADR(TxData[TxLen]));
	TxLen := RAWTOHEX(ADR(INV[Cmd_ObjIdx].FaultData.OpTime),4,ADR(TxData[TxLen]));
	TxLen := RAWTOHEX(ADR(INV[Cmd_ObjIdx].FaultData.InvStatus),2,ADR(TxData[TxLen]));
	TxLen := RAWTOHEX(ADR(INV[Cmd_ObjIdx].FaultData.Vpv_ref),2,ADR(TxData[TxLen]));
	TxLen := RAWTOHEX(ADR(INV[Cmd_ObjIdx].FaultData.Vpv),2,ADR(TxData[TxLen]));
	TxLen := RAWTOHEX(ADR(INV[Cmd_ObjIdx].FaultData.Vmain),2,ADR(TxData[TxLen]));
	TxLen := RAWTOHEX(ADR(INV[Cmd_ObjIdx].FaultData.Status2),2,ADR(TxData[TxLen]));
	TxLen := RAWTOHEX(ADR(INV[Cmd_ObjIdx].FaultData.Status1),2,ADR(TxData[TxLen]));
	TxLen := RAWTOHEX(ADR(INV[Cmd_ObjIdx].FaultData.Tboard),2,ADR(TxData[TxLen]));
	TxLen := RAWTOHEX(ADR(INV[Cmd_ObjIdx].FaultData.Tigbt),2,ADR(TxData[TxLen]));
	TxLen := RAWTOHEX(ADR(INV[Cmd_ObjIdx].FaultData.I_u),2,ADR(TxData[TxLen]));
	TxLen := RAWTOHEX(ADR(INV[Cmd_ObjIdx].FaultData.I_v),2,ADR(TxData[TxLen]));
	TxLen := RAWTOHEX(ADR(INV[Cmd_ObjIdx].FaultData.I_w),2,ADR(TxData[TxLen]));
	TxLen := RAWTOHEX(ADR(INV[Cmd_ObjIdx].FaultData.ClampStatus),2,ADR(TxData[TxLen]));
	TxLen := RAWTOHEX(ADR(INV[Cmd_ObjIdx].FaultData.DigOutput),2,ADR(TxData[TxLen]));
	TxLen := RAWTOHEX(ADR(INV[Cmd_ObjIdx].FaultData.IgbtFault),2,ADR(TxData[TxLen]));
	TxLen := RAWTOHEX(ADR(INV[Cmd_ObjIdx].FaultData.Psupp),4,ADR(TxData[TxLen]));
	TxLen := RAWTOHEX(ADR(INV[Cmd_ObjIdx].FaultData.Epv),4,ADR(TxData[TxLen]));

END_IF
END_ACTION
ACTION Cmd_STR:
(* Check if object index out of range *)
IF Cmd_ObjIdx=0 OR Cmd_ObjIdx>Plant_STR THEN
	Cmd_R:=2;
	RETURN;
END_IF

(* Execute the command only if it equals  0 *)
IF Cmd_C<8 THEN

	STR[Cmd_ObjIdx].FaultAddr := 7711 + Cmd_C * 25;			(* Set right address ModBus of first alarm to be read	*)

	Cmd_RLen := 14;

	TxLen := RAWTOHEX(ADR(STR[Cmd_ObjIdx].FaultData.M018),2,ADR(TxData[TxLen]));
	TxLen := RAWTOHEX(ADR(STR[Cmd_ObjIdx].FaultData.M020),2,ADR(TxData[TxLen]));
	TxLen := RAWTOHEX(ADR(STR[Cmd_ObjIdx].FaultData.Tmodule),2,ADR(TxData[TxLen]));
	TxLen := RAWTOHEX(ADR(STR[Cmd_ObjIdx].FaultData.SuppTime),4,ADR(TxData[TxLen]));
	TxLen := RAWTOHEX(ADR(STR[Cmd_ObjIdx].FaultData.OpTime),4,ADR(TxData[TxLen]));

ELSE

	Cmd_R := 3;

END_IF
END_ACTION
ACTION Cmd_SYS:
(* Check index *)
IF Cmd_ObjIdx<>0 THEN
	Cmd_R:=2;
	RETURN;
END_IF

(* Process command *)
CASE Cmd_C OF

	0: (* ECHO *)
		IF Cmd_CLen<>0 THEN
			TxLen:=0;
		END_IF

	1: (* LOG REQUEST *)
		LogTrig();

	2: (* REARM *)
		Sys.Warning:=FALSE;
		Sys.Alarm:=FALSE;
		Sys.AlarmStop:=FALSE;

	3: (* GET INFO1 *)
		Cmd_RLen:=6;
		TxLen:=TxLen+RAWTOHEX(ADR(Plant_SN),4,ADR(TxData[TxLen]));
		TxLen:=TxLen+RAWTOHEX(ADR(Plant_SW_VER),2,ADR(TxData[TxLen]));

	14: (*  Imposto data e ora del PLC  *)


			Cmd_Buf_U16:=ADR(Cmd_Buf[8]);
			SetAnno:= Cmd_Buf_U16^; 												(* Anno *)
			Cmd_Buf_U16:=ADR(Cmd_Buf[10]);
			SetMese:= Cmd_Buf_U16^;												 	(* mese *)
			Cmd_Buf_U16:=ADR(Cmd_Buf[12]);
			SetGiorno:=( Cmd_Buf_U16^);											 	(* Giorno *)
			Cmd_Buf_U16:=ADR(Cmd_Buf[14]);
			SetOra:=( Cmd_Buf_U16^); 												(* ora *)
			Cmd_Buf_U16:=ADR(Cmd_Buf[16]);
			SetMinuti:= ( Cmd_Buf_U16^);										 	(* Minuti *)
			Cmd_Buf_U16:=ADR(Cmd_Buf[18]);
			SetSecondi:= ( Cmd_Buf_U16^);										 	(* secondi *)

			SysRtcSetTime((SetDataTime(SetAnno,SetMese,SetGiorno,SetOra,SetMinuti,SetSecondi)));

ELSE
	Cmd_R:=3;
END_CASE
END_ACTION
ACTION Command:
(* Default response OK/NODATA *)
Cmd_R:=0;
Cmd_RLen:=0;
TxLen:=16;

(* Check object *)
CASE Cmd_Obj OF

	EO_SYS:
		Cmd_SYS();

	EO_INV:
		Cmd_INV();

	EO_STR:
		Cmd_STR();
ELSE
	Cmd_R:=1;
END_CASE

(* Generate response *)
IF TxLen>0 THEN
	RAWTOHEX(ADR(Cmd_Obj)	,2,ADR(TxData[ 0]));
	RAWTOHEX(ADR(Cmd_ObjIdx),2,ADR(TxData[ 4]));
	RAWTOHEX(ADR(Cmd_R)		,2,ADR(TxData[ 8]));
	RAWTOHEX(ADR(Cmd_RLen)	,2,ADR(TxData[12]));
	TxTrig:=TRUE;
END_IF
END_ACTION

(* POU Utils Functions/TCPSERVER, ST *)
FUNCTION_BLOCK TCPSERVER
(***********************************************************************************************************	*)
(* Version: 1.6                                    			          											*)
(* Date: 11.02.2011                                   					          							    *)
(***********************************************************************************************************	*)
(* WAGO Kontakttechnik GmbH Hansastr. 27 32423 Minden(Westf.)													*)
(* Tel. +0049 571/887-0 Fax. +0049 571/887-0																	*)
(* Author: VB																									*)
(***********************************************************************************************************	*)
(*Description:	A TCP server to read and write data													       		*)
(*Historie:																										*)
(*Version 1.6: 11.02.2011: Changes according to 750-880/881											 			*)
(*Version 1.5: 27.11.2008 Bugfix allow reuse port																*)
(*Version 1.4: 13.10.2008 Bugfix transmitting large data														*)
(*Version 1.3: 15.01.2007 Changes according to FW11																*)
(*Version 1.2: 09.03.2006 Changes for socket handle 0											       			*)
(*Version 1.1: 14.02.2005 Release																				*)
(***********************************************************************************************************	*)
VAR CONSTANT
	STATE_INIT     				 : BYTE:= 0;
	STATE_OPEN     				 : BYTE:= 1;
	STATE_TX       				 : BYTE:= 20;
	STATE_RX       				 : BYTE:= 30;
	STATE_CLOSE    				 : BYTE:= 40;
	STATE_ERROR_TRAP		 	 : BYTE:= 200;
END_VAR
VAR_INPUT
	xEnable    					: BOOL;	 (* Set TRUE to enable function block *)
	wPortNumber					: WORD;  (* Port *)
	tServerTimeOut				: TIME:=t#50s;
	ptSendData					: POINTER TO ARRAY[0..MAX_SEND_TCP_SERVER] OF BYTE;
	diSendCount					: DINT;
END_VAR
VAR_OUTPUT
	xClientConnected  			: BOOL:= FALSE;
	diError 					: DINT:= 0;
END_VAR
(* Status Codes -----------------------------------------
	16#8001 => No socket descriptor available 
	16#8002 => SysSockBind fails 
	16#8003 => SysSockListen fails 
	16#8004 => switching to none blocking mode fails
	16#8005 => SysSockClose() returns FALSE 
    16#8006 => SysSockConnect() fails
    16#8007 => SysSockSend() fails
	16#8008 => error state machine 
	16#8009 => timeout while waiting for data from server 
	16#0001 => server waiting for client to establish connection
------------------------------------------------------------*)
VAR_IN_OUT
	xStartSend					: BOOL;
	aReceiveBuffer				: ARRAY [0..MAX_RECEIVE_TCP_SERVER] OF BYTE;
	diReceiveCount				: DINT;
END_VAR

VAR
	m_State    					: BYTE:= 0;
	m_ReceiveBuffer				: ARRAY [0..MAX_RECEIVE_TCP_SERVER_SOCKET] OF BYTE;
	m_ServerSocket				: DINT:= SOCKET_INVALID;
	m_Socket					: DINT:= SOCKET_INVALID;
	m_AddressInfo				: SOCKADDRESS;
	m_BytesReceived				: DINT;
	m_diReturn					: DINT;
	m_xReturn					: BOOL;
	m_SizeSockadr				: DWORD;
	m_ConnectionWatchdog		: TON;
	m_Flags						: DINT;
	m_NoneBlocking   			: DINT:= 1;
	m_Blocking   				: DINT:= 0;
	i							: INT;
	m_count						: DINT;
	diOption					: DINT := 1;
	on: DINT;
END_VAR
IF xEnable THEN
	CASE m_State OF
		STATE_INIT:
			(* Create Socket *)
			m_ServerSocket:= SysSockCreate( SOCKET_AF_INET, SOCKET_STREAM, 0);
			IF m_ServerSocket = SOCKET_INVALID THEN
				(* *)
				diError:= 16#8001;
				m_State:= STATE_ERROR_TRAP;
				RETURN;
			ELSE
				;
			END_IF
			(* Address bindings *)
			(********************)
			on:=1;
			SysSockSetOption( m_ServerSocket, SOCKET_SOL, SOCKET_SO_REUSEADDR, ADR(on), SIZEOF(on) );

			m_AddressInfo.sin_family:= SOCKET_AF_INET;
			m_AddressInfo.sin_port  := SysSockHtons( wPortNumber);
			m_AddressInfo.sin_addr  := SOCKET_INADDR_ANY;
			IF NOT SysSockBind( m_ServerSocket, ADR(m_AddressInfo), SIZEOF(m_AddressInfo)) THEN
				diError:= 16#8002;
				m_State:= STATE_ERROR_TRAP;
				RETURN;
			END_IF
			(* Wait for connections *)
			(************************)
			IF NOT SysSockListen( m_ServerSocket, 1) THEN
				diError:= 16#8003;
				m_State:= STATE_ERROR_TRAP;
			END_IF

			(* Puts SOCKET in NonBlocking mode *)
			m_diReturn:= SysSockIoctl( m_ServerSocket, SOCKET_FIONBIO, ADR(m_NoneBlocking));

			m_State:= STATE_OPEN;


		STATE_OPEN: 	(* Waiting for incomming connection *)
				m_SizeSockadr:=SIZEOF(m_AddressInfo);
				m_Socket:= SysSockAccept( m_ServerSocket, ADR(m_AddressInfo), ADR(m_SizeSockadr));
				diError:=State_open;
				IF m_Socket <> SOCKET_INVALID THEN
					xClientConnected:=TRUE;
					(*Set Push-Bit:new V1.5*)
					IF ADR(%MW0)=16#30000000  OR ADR(%MW0)=16#20000000 THEN (*841 or 881*)
						SysSockSetOption(
							diSocket:=m_Socket,
							diLevel:=6,
							diOption:=SOCKET_TCP_NODELAY,
							pOptionValue:=ADR(diOption),
							diOptionLength:=SIZEOF(diOption));
					ELSE
							;
					END_IF
					SysSockIoctl( m_Socket, SOCKET_FIONBIO, ADR(m_NoneBlocking));
					m_State:= STATE_RX;
					diError:=0;
				END_IF

		STATE_RX:
					m_BytesReceived:= SysSockRecv( m_Socket, ADR(m_ReceiveBuffer), SIZEOF(m_ReceiveBuffer), 0);
					CASE m_BytesReceived OF
					-1:(*no data available or error occured*)
						m_ConnectionWatchdog(IN:=TRUE , PT:=tServerTimeOut );
						IF m_connectionWatchdog.Q THEN
							m_State:= STATE_CLOSE;
							m_ConnectionWatchdog(IN:=FALSE);(*reset connection watchdog*)
							diError := 16#8009;
						END_IF
					0:(* socket was "gracefully closed"  *)
						m_State:= STATE_CLOSE;
						diError := 16#8003;
					ELSE
						(* Copy received data into receive buffer *)
						(********************************)
						FOR i:= 0 TO DINT_TO_INT(m_BytesReceived	)-1 DO
							aReceiveBuffer[diReceiveCount]:= m_ReceiveBuffer[i];
							diReceiveCount:=(diReceiveCount+1) MOD SIZEOF(aReceiveBuffer);
						END_FOR

						m_ConnectionWatchdog(IN:=FALSE);(*reset connection watchdog*)
					END_CASE

				(*send data*)
				IF xStartSend	 THEN
					m_State := STATE_TX;
				END_IF

	STATE_TX:	 (* send TCP-message *)
		m_diReturn := SysSockSend(diSocket := m_Socket,
								  pbyBuffer := ADR(ptSendData^[m_count]),(*geändert V1.4 bisher: [0] *)
								  diBufferSize := diSendCount-m_count,
								  diFlags :=m_Flags);
		CASE m_diReturn OF
		-1:	(* ERROR or data could not yet be send (V1.3 due to new FW11) *)
			m_ConnectionWatchdog(IN:=TRUE , PT:=tServerTimeOut );
			IF m_connectionWatchdog.Q THEN
				m_State:= STATE_CLOSE;
				m_ConnectionWatchdog(IN:=FALSE);(*reset connection watchdog*)
				diError := 16#8007;
			END_IF
		0: (* socket was "gracefully closed"  *)
			m_State := STATE_CLOSE;
			diError := 16#8003;
		ELSE (* succesful *)
			m_count:=m_count+m_diReturn;
			IF m_count>=diSendCount THEN
				diError := 16#0000;
				m_State := STATE_RX;
				m_count:=0;
				xStartSend:=FALSE;
			END_IF
			m_ConnectionWatchdog(IN:=FALSE);(*reset connection watchdog*)
		END_CASE


		STATE_CLOSE:	(* Close the server *)

		IF ADR(%MW0)=16#30000000  OR ADR(%MW0)=16#20000000 THEN (*841 or 881*)
			;
		ELSE
			IF m_Socket>=0 THEN
				SysSockShutdown(m_Socket, 0);;(*870*)
			END_IF
		END_IF
		IF m_Socket>=0 THEN
			SysSockClose( m_Socket);
		END_IF
		xClientConnected:= FALSE;
		m_State:= STATE_OPEN; (* Try to open the server again *)
		m_ConnectionWatchdog(IN:=FALSE);(*reset connection watchdog*)

		STATE_ERROR_TRAP: (* Error Read/Write socket  *)
			m_State:= STATE_ERROR_TRAP;

	ELSE  (* Bad FSM code trap  *)
			m_State:= STATE_ERROR_TRAP;
			diError:= 16#8008;
	END_CASE;
ELSE
	IF m_State <> STATE_INIT THEN
		IF ADR(%MW0)=16#30000000  OR ADR(%MW0)=16#20000000 THEN (*841 or 881*)
			;
		ELSE
			IF m_Socket>=0 THEN
				SysSockShutdown(m_Socket, 0);;(*870*)
			END_IF
		END_IF
		IF m_Socket>=0 THEN
			SysSockClose( m_Socket);
		END_IF
		IF ADR(%MW0)=16#30000000  OR ADR(%MW0)=16#20000000 THEN (*841 or 881*)
			;
		ELSE
			IF m_ServerSocket>=0 THEN
				SysSockShutdown(m_ServerSocket, 0);;(*870*)
			END_IF
		END_IF
		IF m_ServerSocket>=0 THEN
			SysSockClose( m_ServerSocket);
		END_IF
		xClientConnected:= FALSE;
		diError:= 0;
		m_State:= STATE_init; (* Try to open the server again *)
		m_ConnectionWatchdog(IN:=FALSE);(*reset connection watchdog*)
	END_IF
END_IF
END_FUNCTION_BLOCK

(* POU Utils Functions/HEXTORAW, ST *)
FUNCTION HEXTORAW : WORD
VAR_INPUT
	pString		: POINTER TO BYTE;
	StringLen	: WORD;
	pData		: POINTER TO BYTE;
END_VAR
VAR
	xl: WORD;
	xi: WORD;
	xr: BYTE;
END_VAR
(* Convert transmitted hexadecimal data, encoded as string, back to hexadecimal format (see ASCII vs Hex table) *)
xl:=0;
xi:=0;

WHILE xi<StringLen DO

	IF pString^>=97 AND pString^<=102 THEN		(* Lower case letter "a..f" *)
		xr := pString^ - 87;
	ELSIF pString^>=65 AND pString^<=70 THEN	(* Upper case letter "A..F" *)
		xr := pString^ - 55;
	ELSIF pString^>=48 AND pString^<=57 THEN	(* Digit "0..9" *)
		xr := pString^ - 48;
	ELSE
		xr := 16;
	END_IF

	IF xr<16 THEN
		IF (xi AND 1)=0 THEN					(* Enter this if when even index (last digit is 0) *)
			pData^ := xr * 16;
		ELSE
			pData^ := pData^ + xr;				(* Enter this else when odd index (last digit is 1) *)
			pData := pData + 1;
			xl := xl + 1;
		END_IF
	END_IF

	xi := xi + 1;
	pString := pString + 1;

END_WHILE

HEXTORAW:=xl;									(* Number of word *)

(* NB Byte are transmitted MSB first *)
END_FUNCTION

(* POU Utils Functions/RAWTOHEX, ST *)
FUNCTION RAWTOHEX : WORD
VAR_INPUT
	pData: POINTER TO BYTE;
	DataLen: WORD;
	pString: POINTER TO BYTE;
END_VAR
VAR
	xl: WORD;
END_VAR
xl:=0;

WHILE DataLen>0 DO

	pString^ := (pData^ / 16#10) + 48 + (((pData^ / 16#10)/10)*7);
	pString:=pString+1;
	pString^ := (pData^ AND 16#0F)  + 48 + (((pData^ AND 16#0F)/10)*7);
	pString:=pString+1;
	pData:=pData+1;
	DataLen:=DataLen-1;
	xl:=xl+2;

END_WHILE

(*pString^:=0;*)

RAWTOHEX:=xl;
END_FUNCTION

(* POU Utils Functions/SetDataTime, ST *)
FUNCTION SetDataTime : DT
VAR_INPUT
	year : INT;
	month : INT;
	day : INT;
	hour : INT;
	minute : INT;
	second : INT;
END_VAR

VAR
	count : INT;
END_VAR
(* Creazione variabiletipo DT per creare Orario da dare al PLC *)


IF month > 2 THEN
	count := (month - 1) * 30;
	IF month > 7 THEN count := count + SHR(month - 3,1); ELSE count := count + SHR(month - 4,1); END_IF;
	(* chech for leap year and add one day if true *)
	IF SHL(year,14) = 0 THEN count := count + 1; END_IF;
ELSE
	count := (month - 1) * 31;
END_IF;


SetDataTime := DWORD_TO_DT(DATE_TO_DWORD( DWORD_TO_DATE((INT_TO_DWORD(count + day - 1) + SHR(INT_TO_DWORD(year) * 1461 - 2878169, 2)) * 86400))
				+ INT_TO_DWORD(SECOND)
				+ INT_TO_DWORD(MINUTE) * 60
				+ INT_TO_DWORD(HOUR) * 3600);
END_FUNCTION

(* POU Utils/CSV_Log, ST *)
FUNCTION CSV_Log : BOOL
VAR_INPUT
END_VAR
VAR CONSTANT
	LogFileName:STRING:='S:\LOGS_ID4V3.CSV';
END_VAR
VAR
	s1 : STRING(256);
	hFile: 	DWORD;
END_VAR
(* Check file presence *)
hFile:=SysFileOpen(LogFileName,'r');
IF hFile=0 THEN
	(*** File not exist *** Create file and write header *)
	hFile:=SysFileOpen(LogFileName,'w');
	IF hFile<>0 THEN
		(* Write CSV header *)
		s1:='Title1;Title2,...';
		SysFileWrite(hFile, ADR(s1), LEN(s1));
		SysFileWrite(hFile, ADR(Logger_CRLF), LEN(Logger_CRLF));	(* End of line encoding	*)
	END_IF
ELSE
	(*** File exist *** Close file and reopen in append mode *)
	SysFileClose(hFile);
	hFile:=SysFileOpen(LogFileName,'a');
END_IF

(* Log to file *)
IF hFile<>0 THEN
	(* Date stamp *)
	s1:=REPLACE( Sys.Time_LogString , ' ' , 1 , 11 );
	SysFileWrite(hFile, ADR(s1), LEN(s1));
	(* Write CSV data *)
	s1:=CONCAT(';', 'Data1' );
	s1:=CONCAT(s1 , ';');
	s1:=CONCAT(s1 , 'Data2' );
	s1:=CONCAT(s1 , ';');
	s1:=CONCAT(s1 , '...' );
	SysFileWrite(hFile, ADR(s1), LEN(s1));
	(* Add line CRLF and close *)
	SysFileWrite(hFile, ADR(Logger_CRLF), LEN(Logger_CRLF));
	SysFileClose(hFile);
END_IF
END_FUNCTION

(* POU PLC_SYS_FAST, ST *)
PROGRAM PLC_SYS_FAST
VAR
END_VAR
IF Sys.Status = S_RUNNING THEN

	SYS_Proc();
	SWI_Proc();

END_IF
END_PROGRAM

(* POU Plant/SYS_Proc, ST *)
PROGRAM SYS_Proc
VAR
(*	fALARM_PB		:FLT_TAP;
	fALARM_TB		:FLT_TAP;
	fALARM_PM		:FLT_TAP; *)

(*	fGZB_ST			:FLT_TAP;  (* GATEWAY ZIGBEE *)*)
(*	fVPN_ST1		:FLT_TAP;  (* VPN CONNECT *)*)
	fVPN_ST2		:FLT_TAP;  (* VPN STATUS *)
(*	fKEY_CT_ST		:FLT_TAP;  (* DOOR1 *)*)
(*	fKEY_SCT_ST		:FLT_TAP;  (* DOOR2 *)*)
	fKEY_QE_ST		:FLT_TAP;  (* DOOR3 *)

END_VAR
(*************** ISPESL *****************)
(*
fALARM_PB(IN:=ALARM_PB);
IF fALARM_PB.EVH THEN
	LogEv(EL_AlarmStop,EO_PBV,1,1,'Over_Pressure_Alarm');
END_IF

fALARM_TB(IN:=ALARM_TB);
IF fALARM_TB.EVH THEN
	LogEv(EL_AlarmStop,EO_TBV,1,1,'Over_Temperature_Alarm');
END_IF

fALARM_PM(IN:=ALARM_PM);
IF fALARM_PM.EVH THEN
	LogEv(EL_AlarmStop,EO_PMV,1,1,'Under_Pressure_Alarm');
END_IF
*)
(****************************************)

(*### VPN Connection Check ###*)(*
fVPN_ST1(IN:=VPN_ST1);
IF fVPN_ST1.EVH THEN
	LogEv(EL_Log,EO_VPN,1,1,'CONNECT_ON');
END_IF
IF fVPN_ST1.EVL THEN
	LogEv(EL_Log,EO_VPN,1,2,'CONNECT_OFF');
END_IF*)

(*### VPN Status Check ###*)
fVPN_ST2(IN:=VPN_ST2);
IF fVPN_ST2.EVH THEN
	LogEv(EL_Log,EO_VPN,1,3,'STATUS_UP');
END_IF
IF fVPN_ST2.EVL THEN
	LogEv(EL_Wrn,EO_VPN,1,4,'STATUS_DOWN');
END_IF

(*### DOOR01 Status Check ###*)(*
fKEY_CT_ST(IN:=KEY_CT_ST);
IF fKEY_CT_ST.EVH THEN
	LogEv(EL_Log,EO_DOOR,1,2,'Centrale_termica_Close');
END_IF
IF fKEY_CT_ST.EVL THEN
	LogEv(EL_Wrn,EO_DOOR,1,1,'Centrale_termica_Open');
END_IF*)

(*### DOOR02 Status Check ###*)(*
fKEY_SCT_ST(IN:=KEY_SCT_ST);
IF fKEY_SCT_ST.EVH THEN
	LogEv(EL_Log,EO_DOOR,2,2,'Sottocentrale_termica_Close');
END_IF
IF fKEY_SCT_ST.EVL THEN
	LogEv(EL_Wrn,EO_DOOR,2,1,'Sottocentrale_termica_Open');
END_IF*)

(*### DOOR03 Status Check ###*)
fKEY_QE_ST(IN:=KEY_QE_ST);
IF fKEY_QE_ST.EVH THEN
	LogEv(EL_Log,EO_DOOR,3,2,'Quadro_Close');
END_IF
IF fKEY_QE_ST.EVL THEN
	LogEv(EL_Wrn,EO_DOOR,3,1,'Quadro_Open');
END_IF
END_PROGRAM

(* POU Utils Functions/FLT_TAP, ST *)
FUNCTION_BLOCK FLT_TAP
VAR_INPUT
	IN		: BOOL;
	TAP		: BYTE:=4;
	INITEV	: BOOL:=TRUE;
END_VAR
VAR_OUTPUT
	OUT		: BOOL;
	EVH		: BOOL;
	EVL		: BOOL;
END_VAR
VAR
	init	: BOOL:=FALSE;
	cnt		: BYTE;
END_VAR
EVH:=FALSE;
EVL:=FALSE;

(* This first IF is done only the first time the FB is called, to read the actual (startup) value of the element;
   After first iteration, "init" becomes true and this IF is always skipped, unless a reset occurs	*)
IF NOT init THEN
	init := TRUE;
	IF INITEV THEN
		OUT  := NOT IN;
		cnt  := TAP;
	ELSE
		OUT  := IN;
	END_IF
END_IF

(* Need "TAP" equals level before update "OUT"	*)
IF OUT<>IN THEN
	cnt:=cnt+1;
	IF cnt>TAP THEN
		OUT:=IN;
		cnt:=0;
		IF OUT THEN EVH:=TRUE; ELSE EVL:=TRUE; END_IF
	END_IF
ELSE
	cnt:=0;
END_IF
END_FUNCTION_BLOCK

(* POU TCP_Logger/LogEv, ST *)
FUNCTION LogEv : BOOL
VAR_INPUT
	Level	: en_Logger_ErrLev;
	Object  : en_SYS_Objects;
	Index	: WORD;
	Error	: WORD;
	Message : STRING;
END_VAR
VAR
	s1 : STRING(160);
	i  : INT;
END_VAR
(* Generates the log for the error revealed	*)

(* Execute error level operations *)
CASE Level OF
	EL_Wrn: 		Sys.Warning:=TRUE;
	EL_Alarm: 		Sys.Alarm  :=TRUE;
	EL_AlarmStop: 	Sys.Alarm  :=TRUE; (* GO TO STOP STATE!! *)
END_CASE

(*** Runtime memory for last 5 logs (it's a sort of backup)	***)
(* Fill lastlog list *)
s1:=CONCAT(Sys.Time_LogString,';Lev=');			(* Insert current data and time read at the beginning *)
s1:=CONCAT(s1,INT_TO_STRING(Level));			(* Insert error level	*)
s1:=CONCAT(s1,';Obj=');
s1:=CONCAT(s1,INT_TO_STRING(Object));			(* Insert object who generates the error	*)
s1:=CONCAT(s1,';Idx=');
s1:=CONCAT(s1,WORD_TO_STRING(Index));			(* Insert ID of the object in the system	*)
s1:=CONCAT(s1,';Err=');
s1:=CONCAT(s1,WORD_TO_STRING(Error));			(* Insert specific error	*)

(* This is used to keep last 5 logs in memory	*)
Sys.LastLogs_Dat[Sys.LastLogs_Idx]:=s1;
Sys.LastLogs_Msg[Sys.LastLogs_Idx]:=Message;
Sys.LastLogs_Idx:=Sys.LastLogs_Idx+1;

IF Sys.LastLogs_Idx>5 THEN Sys.LastLogs_Idx:=0; END_IF	(* If log index reach the end of the array, restart the index (Set it to 0)	*)

(*---------------------------------------------------------------*)
	Logger_Head();
(*---------------------------------------------------------------*)

(* Insert ERR *)		(* Repeat previous steps to create the log has to be transmitted on the network	*)
IF Level = EL_Evt THEN
	s1:=CONCAT('&EVT=',INT_TO_STRING(Level-EL_Evt));
ELSE
	s1:=CONCAT('&ERR=',INT_TO_STRING(Level));
END_IF
s1:=CONCAT(s1,';');
s1:=CONCAT(s1,INT_TO_STRING(Object));
s1:=CONCAT(s1,';');
s1:=CONCAT(s1,WORD_TO_STRING(Index));
s1:=CONCAT(s1,';');
s1:=CONCAT(s1,WORD_TO_STRING(Error));
s1:=CONCAT(s1,';');

ADDSTRING(ADR(Logger.TData), ADR(s1), Logger.TLen);		(* Add this part of the log to the previous one (the header)	*)
s1:=Message;
STR_NOSPACES(ADR(s1));									(* Check there are no blank spaces in the "Message"	*)
ADDSTRING(ADR(Logger.TData), ADR(s1), Logger.TLen);		(* Add error message to the rest of the log file	*)

(*---------------------------------------------------------------*)
	Logger_Send();
(*---------------------------------------------------------------*)
END_FUNCTION

(* POU TCP_Logger/Logger_Head, ST *)
FUNCTION Logger_Head : BOOL
VAR
	s1 : STRING(160);
	i  : BYTE;
END_VAR
(* Create the header to transmit the logfile on the VPN according to internal protocol	*)
Logger.TLen:=0;

(* Set GET header *)
ADDSTRING(ADR(Logger.TData), ADR(Logger_GETSTART), Logger.TLen);

(* Insert Header *)
s1:=INSERT('ID=&V=1&D=',DWORD_TO_STRING(Plant_SN),3);		(* Insert plant ID after 3 characters, therefore after string
																'ID='	*)
s1:=CONCAT(s1,Sys.Time_LogString);							(* Add Data and Time	*)
s1:=CONCAT(s1,'&S=');

(* Check what to signal according to the flag: Alarm, Warning or everything OK	*)
IF Sys.Alarm THEN i:=2; ELSIF Sys.Warning THEN i:=1; ELSE i:=0; END_IF
s1:=CONCAT(s1,BYTE_TO_STRING(i));

ADDSTRING(ADR(Logger.TData), ADR(s1), Logger.TLen);
END_FUNCTION

(* POU Utils Functions/ADDSTRING, ST *)
FUNCTION ADDSTRING : BOOL (* Append string to a byte buffer *)
VAR_INPUT
	pTxData: POINTER TO BYTE;
	pString: POINTER TO BYTE;
END_VAR
VAR_IN_OUT
	TxLen: DINT;
END_VAR
VAR
END_VAR
(* Add a string starting from an offset ("TxLen") using pointer. Stop the add when the string to copy has a 0 as argument	*)
pTxData:=pTxData+TxLen;
WHILE pString^<>0 DO
	pTxData^:=pString^;
	pString:=pString+1;
	pTxData:=pTxData+1;
	TxLen:=TxLen+1;
END_WHILE
END_FUNCTION

(* POU Utils Functions/STR_NOSPACES, ST *)
FUNCTION STR_NOSPACES : BOOL (* Replace spaces and bad chars with allowed ones, used as HTTP-GET validator *)
VAR_INPUT
	pString: POINTER TO BYTE;
END_VAR
VAR
END_VAR
WHILE pString^<>0 DO
	IF pString^=16#20 (* space *) THEN pString^:=16#5F; (*'_'*) END_IF
	pString:=pString+1;
END_WHILE
END_FUNCTION

(* POU TCP_Logger/Logger_Send, ST *)
FUNCTION Logger_Send : BOOL
VAR
	hFile: 	DWORD;
	pos:	DWORD;
END_VAR
(* Finalize string *)
ADDSTRING(ADR(Logger.TData), ADR(Logger_GETEND), Logger.TLen);		(* Code that identifies the end of the "GET" log  *)

(* Read log position *)
pos:=SysFileGetSize(Logger_DataFile);								(* Get size in byte of the file	*)

(* Check log size, bckup and erase if no pending messages *)
IF pos>5000000(*5M*) THEN
	hFile:=SysFileOpen(Logger_IndexFile,'r');

	IF hFile=0 THEN							(* If "Logger_IndexFile" doesn't exist -> No pending messagge to be transmitted	*)
		SysFileDelete(Logger_DataFileOld);							(* Delete old log file (backup)	*)
		SysFileRename(Logger_DataFile,Logger_DataFileOld);			(* Rename new log file as "DataFileOld" (backup) *)
		pos:=0;
	ELSE
		SysFileClose(hFile);
	END_IF
END_IF
(* ^^^ Delete old backup file and if actual logger file is too big and all messagges have been transmitted, set it as backup *)

(* Write message on log file *)
hFile:=SysFileOpen(Logger_DataFile,'a');							(* Open in write mode, but new data ar added at the end *)

(* If no error occurs when opening the log file, write new data ("Logger.TData")	*)
IF hFile<>0 THEN
	SysFileWrite(hFile, ADR(Logger.TData), Logger.TLen);
	SysFileClose(hFile);
ELSE
	Sys.Warning:=TRUE;		(* Set a system warning	*)
END_IF


(* Check logger status *)
IF Logger.SendReq=FALSE THEN
	(* Set log position for recovery *)
	Logger.SendIdx:=pos;
	(* Copy message data *)
	MEMCPY(ADR(Logger.TData),ADR(Logger.SendData),DINT_TO_WORD(Logger.TLen));
	Logger.SendLen:=Logger.TLen;
	(* Trigger request *)
	Logger.SendReq:=TRUE;
ELSE
	(* Connection still busy, so it's not possible to send now data. Write the LoggerIndex file	*)
	(* Add message position+size in recovery indexes *)
	hFile:=SysFileOpen(Logger_IndexFile,'a');
	SysFileWrite(hFile, ADR(pos), SIZEOF(pos));
	SysFileWrite(hFile, ADR(Logger.TLen), SIZEOF(Logger.TLen));
	SysFileClose(hFile);
END_IF
END_FUNCTION

(* POU Utils Functions/MEMCPY, ST *)
FUNCTION MEMCPY:BOOL
VAR_INPUT
	pSourceAddress:POINTER TO ARRAY[1..2] OF BYTE;
	pDestinationAddress:POINTER TO ARRAY[1..2] OF BYTE;
	BytesToCopy:WORD;
END_VAR
VAR
END_VAR
WHILE (BytesToCopy > 0) DO
	pDestinationAddress^[1]:=pSourceAddress^[1]; (* copy bytes from source to destination *)
	pDestinationAddress:=ADR(pDestinationAddress^[2]); (* increment destination *)
	pSourceAddress:=ADR(pSourceAddress^[2]);(* increment source *)
	BytesToCopy:=BytesToCopy -1; (* decrement number of bytes to copy *)
END_WHILE
END_FUNCTION

(* POU Plant/SWI_Proc, ST *)
(*** USE FOR PHOTOVOLTAIC FIELD ***)
PROGRAM SWI_Proc
VAR
		fKEY_QE_MS	:	FLT_TAP;	(* Main switch in the general switchboard *)
		fKEY_QE_MIS	:	FLT_TAP;	(* Main interface switch in the general switchboard	*)
END_VAR
(*** Main switch and Main interface switch managing ***)
(* Ensure inverters are connected to the mains	*)

(* Check main switch	*)
fKEY_QE_MS(IN:= INT01);

IF fKEY_QE_MS.EVH THEN
	LogEv(EL_Log,EO_SWITCH,1,2,'Main_switch_On');			(* It works fine	*)
END_IF
IF fKEY_QE_MS.EVL THEN
	LogEv(EL_Alarm,EO_SWITCH,1,1,'Main_switch_Off');		(* Main switch is off -->> Alarm	*)
END_IF

(* Check main interface switch	*)
fKEY_QE_MIS(IN:= INT02);

IF fKEY_QE_MIS.EVH THEN
	LogEv(EL_Log,EO_SWITCH,2,2,'Main_Interface_On');			(* It works fine	*)
END_IF
IF fKEY_QE_MIS.EVL THEN
	LogEv(EL_Alarm,EO_SWITCH,2,1,'Main_Interface_Off');		(* Main interface is off -->> Alarm	*)
END_IF
END_PROGRAM

(* POU Utils/RTC_Update, ST *)
PROGRAM RTC_Update
VAR
	T: DT;
	TS: STRING;
	TS2: STRING;
	Hour: BYTE;
	Minute: BYTE;
END_VAR
(* Get RTC time *)
T:=SysRtcGetTime(TRUE);
Sys.Time_CT_DT:=T;

(* Calculate variables *)
TS:=DT_TO_STRING(T);								(* Convert a format DATA_AND_TIME into a string, with the following
														result: 'DT#YYYY-MM-DD-HH:MM'	*)

Sys.Time_LogString:=DELETE(STR:=TS, LEN:=3, POS:=1);	(* Delete 3 characters starting from character number 1, the first
															so it deletes 'DT#'	*)

(* Proceed as before to isolate Year, Month and Day and convert them into a number format	*)
TS2:=MID(STR:=TS, LEN:=4, POS:= 4); Sys.Time_Year 	:=STRING_TO_WORD(TS2);
TS2:=MID(STR:=TS, LEN:=2, POS:= 9); Sys.Time_Month	:=STRING_TO_BYTE(TS2);
TS2:=MID(STR:=TS, LEN:=2, POS:=12); Sys.Time_Day  	:=STRING_TO_BYTE(TS2);

Sys.Time_CT_Day:=(32*(Sys.Time_Month-1)+Sys.Time_Day-1);

(* Proceed as before to isolate Hour and minute and convert them into a number format	*)
TS2:=MID(STR:=TS, LEN:=2, POS:=15); Hour			:=STRING_TO_BYTE(TS2);
TS2:=MID(STR:=TS, LEN:=2, POS:=18); Minute		 	:=STRING_TO_BYTE(TS2);

(* Calculate quarters of hour	*)
Sys.Time_CT_Quarter:=Hour*4+(Minute/15);
END_PROGRAM

(* POU Configuration/MODBUS_CONFIGURATION, ST *)
PROGRAM MODBUS_CONFIGURATION        
VAR                                
END_VAR                            
(*                                 
   <?xml version="1.0" encoding="UTF-16" standalone="yes"?>
<network xml_structure_version="1" xml_feature_version="1">
	<generator_settings minRTUTaskCycleTimeMs="5" minEthaskCycleTimeMs="5" ethSlaveMultiplier="0.1" rtuInterfaceMultiplier="0.1" taskGeneration="false"/>
</network>
                              
*)                                 
;                                  
END_PROGRAM

(* POU PLC_WDT, ST *)
PROGRAM PLC_WDT
VAR
END_VAR
LogEv(EL_AlarmStop,EO_SYS,1,10,'Watchdog_expired');
END_PROGRAM

(* POU Utils/USRLED_Update, ST *)
PROGRAM USRLED_Update
VAR
	Status	:	BYTE;
END_VAR
Status := PlantStatus;
PlantStatus := 0;	(* Reset value *)

(* Plant status (Alarm, warning or everything ok) *)
IF Status = 2 THEN
	LED_SET_STATIC(diLed_No:=7, eColor:=2);
	RETURN;
ELSIF Status = 1 THEN
	LED_SET_BLINK(diLed_No:=7, timTime1:=T#500ms, timTime2:=T#500ms, eColor1:=0, eColor2:=3);
	RETURN;
END_IF

(* VPN status led signalling *)
IF VPN_ST2 = 0 THEN
	LED_SET_BLINK(diLed_No:=7, timTime1:=T#500ms, timTime2:=T#500ms, eColor1:=0, eColor2:=2);
	RETURN;
END_IF

(* ModBus status led signalling *)
IF MODB01.MB_MASTER.bInterfaceError <> 0 THEN
	LED_SET_BLINK(diLed_No:=7, timTime1:=T#1s, timTime2:=T#1s, eColor1:=0, eColor2:=2);
	RETURN;
END_IF

(* Main Siwtch or Interface *)
IF INT01 = 0 OR INT02 = 0 THEN
	LED_SET_BLINK(diLed_No:=7, timTime1:=T#2s, timTime2:=T#2s, eColor1:=0, eColor2:=2);
	RETURN;
END_IF

(* System status led signalling *)
CASE SYS.Status OF

	S_STARTUP:
				(* Orange static *)
				LED_SET_STATIC(diLED_No:=7, eColor:=3);

	S_RUNNING:
				(* Green static *)
				LED_SET_STATIC(diLED_No:=7, eColor:=1);

END_CASE
END_PROGRAM

(* POU Utils Functions/AVERAGE_DINT, ST *)
FUNCTION_BLOCK AVERAGE_DINT
VAR_INPUT
	IN: 	DINT;
END_VAR
VAR_OUTPUT
	HI:		DINT;
	AVG:	DINT;
	LOW:	DINT;
	ERR:	BOOL;
END_VAR
VAR
	sum:	REAL;
	cnt:	WORD;
END_VAR
IF cnt>=65000 THEN
	ERR:=TRUE;
	Read();
	sum := sum - DINT_TO_REAL(AVG);
	cnt := cnt - 1;
END_IF

sum := sum + DINT_TO_REAL(IN);
cnt := cnt + 1;

IF IN<LOW THEN LOW:=IN; END_IF
IF IN>HI  THEN HI :=IN; END_IF
END_FUNCTION_BLOCK
ACTION Read:
AVG := REAL_TO_DINT(sum/cnt);
END_ACTION
ACTION Reset:
HI:=IN;
AVG:=IN;
LOW:=IN;
ERR:=FALSE;

sum:=DINT_TO_REAL(IN);
cnt:=1;
END_ACTION

(* POU Utils Functions/AVERAGE_INT, ST *)
FUNCTION_BLOCK AVERAGE_INT
VAR_INPUT
	IN: 	INT;
END_VAR
VAR_OUTPUT
	HI:		INT;
	AVG:	INT;
	LOW:	INT;
	ERR:	BOOL;
END_VAR
VAR
	sum:	DINT;
	cnt:	WORD;
END_VAR
IF cnt>=65000 THEN
	ERR:=TRUE;
	Read();
	sum := sum - AVG;
	cnt := cnt - 1;
END_IF

sum := sum + IN;
cnt := cnt + 1;

IF IN<LOW THEN LOW:=IN; END_IF
IF IN>HI  THEN HI :=IN; END_IF
END_FUNCTION_BLOCK
ACTION Read:
AVG := DINT_TO_INT(sum/cnt);
END_ACTION
ACTION Reset:
HI:=IN;
AVG:=IN;
LOW:=IN;
ERR:=FALSE;

sum:=IN;
cnt:=1;
END_ACTION

(* POU Utils Functions/AVERAGE_T, ST *)
FUNCTION_BLOCK AVERAGE_T
VAR_INPUT
	IN: 	INT;
END_VAR
VAR_OUTPUT
	HI:		INT;
	AVG:	INT;
	LOW:	INT;
	ERR:	BOOL;
END_VAR
VAR
	sum:	DINT;
	cnt:	WORD;
END_VAR
IF cnt>=65000 THEN
	ERR:=TRUE;
	Read();
	sum := sum - AVG;
	cnt := cnt + 1;
END_IF

sum := sum + IN;
cnt := cnt + 1;

IF IN<LOW THEN  LOW:=IN; END_IF
IF IN>HI  THEN HI :=IN; END_IF
END_FUNCTION_BLOCK
ACTION Read:
AVG := DINT_TO_INT(sum/cnt);
END_ACTION
ACTION Reset:
HI:=IN;
AVG:=IN;
LOW:=IN;
ERR:=FALSE;

sum:=IN;
cnt:=1;
END_ACTION

(* POU Utils Functions/BUILD_16TO32_COPY, ST *)
FUNCTION BUILD_16TO32_COPY : DWORD
VAR_INPUT
		LSW	:	WORD;
		MSW	:	WORD;
END_VAR
VAR
		Op1	:	DWORD;
		Op2	:	DWORD;
END_VAR
Op1  := WORD_TO_DWORD(LSW);

Op2 := WORD_TO_DWORD(MSW);
Op2 := SHL(Op2, 16);

BUILD_16TO32_COPY := Op1 + Op2;
END_FUNCTION

(* POU Utils Functions/CheckPlant, ST *)
FUNCTION CheckPlant : BOOL
VAR_INPUT
		Obj_Status_Log	:	BYTE;
END_VAR
VAR
END_VAR
IF Obj_Status_Log = 0 THEN RETURN; END_IF

IF PlantStatus = 2 THEN RETURN; END_IF

IF PlantStatus = 1 THEN
	IF Obj_Status_Log = 2 THEN
		PlantStatus := 2;
		RETURN;
	END_IF
END_IF

IF PlantStatus = 0 THEN
	PlantStatus := Obj_Status_Log;
	RETURN;
END_IF
END_FUNCTION

(* POU Utils Functions/COPY_32SWAP16, ST *)
FUNCTION COPY_32SWAP16:BOOL
VAR_INPUT
	pSourceAddress		:POINTER TO ARRAY[1..2] OF WORD;
	pDestinationAddress	:POINTER TO ARRAY[1..2] OF WORD;
END_VAR
VAR
END_VAR
pDestinationAddress^[1]:=pSourceAddress^[2];
pDestinationAddress^[2]:=pSourceAddress^[1];
END_FUNCTION

(* POU Utils Functions/FLT_EVENT, ST *)
FUNCTION_BLOCK FLT_EVENT
VAR_INPUT
	IN		: BOOL;
	INITEV	: BOOL:=TRUE;
END_VAR
VAR_OUTPUT
	EVH		: BOOL;
	EVL		: BOOL;
END_VAR
VAR
	init	: BOOL:=FALSE;
	old		: BOOL;
END_VAR
EVH:=FALSE;
EVL:=FALSE;

IF NOT init THEN
	init:=TRUE;
	IF INITEV THEN
		old := NOT IN;
	ELSE
		old := IN;
	END_IF
END_IF

IF old<>IN THEN
	old:=IN;
	IF IN THEN EVH:=TRUE; ELSE EVL:=TRUE; END_IF
END_IF

(* NB: Questo functional block segnala l'EVENTO, NON lo STATO.
	   Infatti se IN non muta lo stato, sia EVL sia EVH rimangono FALSE *)
END_FUNCTION_BLOCK

(* POU Utils Functions/FLT_TIME, ST *)
FUNCTION_BLOCK FLT_TIME
VAR_INPUT
	IN		: BOOL;
	TTAP	: TIME:=T#5s;
	INITEV	: BOOL:=TRUE;
END_VAR
VAR_OUTPUT
	OUT		: BOOL;
	EVH		: BOOL;
	EVL		: BOOL;
END_VAR
VAR
	init	: BOOL:=FALSE;
	timer	: TON;
END_VAR
EVH:=FALSE;
EVL:=FALSE;

IF NOT init THEN
	init := TRUE;
	IF INITEV THEN
		OUT  := NOT IN;
	ELSE
		OUT  := IN;
	END_IF
END_IF

IF OUT<>IN THEN
	timer(IN:=TRUE,PT:=TTAP);
	IF timer.Q THEN
		OUT:=IN;
		timer(IN:=FALSE);
		IF OUT THEN EVH:=TRUE; ELSE EVL:=TRUE; END_IF
	END_IF
ELSE
	timer(IN:=FALSE);
END_IF
END_FUNCTION_BLOCK

(* POU Utils Functions/GETBIT, ST *)
FUNCTION GETBIT : BOOL
VAR_INPUT
		IN		:	DWORD;
		Offset	:	BYTE;
END_VAR
VAR
END_VAR
GETBIT := DWORD_TO_BOOL(IN AND(SHL(DWORD#1,Offset)));
END_FUNCTION

(* POU Utils Functions/LAMP_AL_GENERALE, ST *)
FUNCTION_BLOCK LAMP_AL_GENERALE
VAR_INPUT

	Allarme: BOOL;
	Warning: BOOL;
END_VAR
VAR_OUTPUT
	StatoSistema:BYTE;
	SistemaInAllarme:BOOL;
	SistemaWarning:BOOL;
	AllarmeLampada:BOOL;
END_VAR
VAR
	Lampeggio:BLINK;
END_VAR
IF Allarme THEN       					(* Se Allarme Attivo Luce fissa ON *)
	StatoSistema:=2;
	SistemaInAllarme:=TRUE;
	SistemaWarning:=FALSE;
	AllarmeLampada:=TRUE;
ELSIF Warning THEN					(* Se Allarme Attivo Luce fissa pulse *)
	StatoSistema:=1;
	SistemaInAllarme:=FALSE;
	SistemaWarning:=TRUE;
	Lampeggio(ENABLE:=TRUE , TIMELOW:=t#1s , TIMEHIGH:=t#1s , OUT=>AllarmeLampada );
ELSE
	StatoSistema:=0;
	SistemaInAllarme:=FALSE;
	SistemaWarning:=FALSE;
	AllarmeLampada:=FALSE;
END_IF
END_FUNCTION_BLOCK

(* POU Utils Functions/LINEAR, ST *)
FUNCTION LINEAR : REAL (* Linear interpolation *)
VAR_INPUT
	X_In	: REAL;
	P1_X	: REAL;
	P1_Y	: REAL;
	P2_X	: REAL;
	P2_Y	: REAL;
END_VAR
VAR
END_VAR
LINEAR:=P1_Y+(((P2_Y-P1_Y)*(X_In-P1_X))/(P2_X-P1_X));
END_FUNCTION

(* POU Utils Functions/LINEAR_BAD, ST *)
FUNCTION LINEAR_BAD : INT (* Linear interpolation *)
VAR_INPUT
	PuntoMinX	: INT;
	PuntoMaxX	: INT;
	ValIn		: INT;
	PuntoMinY	: REAL;
	PuntoMaxY	: REAL;
	Decimali	: BYTE;
END_VAR
VAR
	Gain				: REAL;
	PuntoMinX_R			: REAL;
	PuntoMaxX_R			: REAL;
	Linearizzazione_R	: REAL;
END_VAR
PuntoMinX_R:=INT_TO_REAL(PuntoMinX);
PuntoMaxX_R:=INT_TO_REAL(PuntoMaxX);

Gain:=(PuntoMaxX_R-PuntoMinX_R)/(PuntoMaxY-PuntoMinY);	(* Calcolo in guadagno per la linarizzazione *)
Linearizzazione_R:=PuntoMinx+(Gain*(ValIn-PuntoMinY));	(* Ottengo il valore linearizzato *)

LINEAR_BAD:=REAL_TO_INT(Linearizzazione_R*(EXPT(10, Decimali)));  (* Ottengo intero con i decimai voluti *)
END_FUNCTION

(* POU TCP_Logger/LogEv_old, ST *)
FUNCTION LogEv_old : BOOL
VAR_INPUT
	Level	: en_Logger_ErrLev;
	Object  : en_SYS_Objects;
	Index	: WORD;
	Error	: WORD;
	Message : STRING;
END_VAR
VAR
	s1 : STRING(160);
	i  : INT;
END_VAR
(* Generates the log for the error revealed	*)

(* Execute error level operations *)
CASE Level OF
	EL_Wrn: 		Sys.Warning:=TRUE;
	EL_Alarm: 		Sys.Alarm  :=TRUE;
	EL_AlarmStop: 	Sys.Alarm  :=TRUE; (* GO TO STOP STATE!! *)
END_CASE

(*** Runtime memory for last 5 logs (it's a sort of backup)	***)
(* Fill lastlog list *)
s1:=CONCAT(Sys.Time_LogString,';Lev=');			(* Insert current data and time read at the beginning *)
s1:=CONCAT(s1,INT_TO_STRING(Level));			(* Insert error level	*)
s1:=CONCAT(s1,';Obj=');
s1:=CONCAT(s1,INT_TO_STRING(Object));			(* Insert object who generates the error	*)
s1:=CONCAT(s1,';Idx=');
s1:=CONCAT(s1,WORD_TO_STRING(Index));			(* Insert ID of the object in the system	*)
s1:=CONCAT(s1,';Err=');
s1:=CONCAT(s1,WORD_TO_STRING(Error));			(* Insert specific error	*)

(* This is used to keep last 5 logs in memory	*)
Sys.LastLogs_Dat[Sys.LastLogs_Idx]:=s1;
Sys.LastLogs_Msg[Sys.LastLogs_Idx]:=Message;
Sys.LastLogs_Idx:=Sys.LastLogs_Idx+1;

IF Sys.LastLogs_Idx>5 THEN Sys.LastLogs_Idx:=0; END_IF	(* If log index reach the end of the array, restart the index (Set it to 0)	*)

(*---------------------------------------------------------------*)
	Logger_Head();
(*---------------------------------------------------------------*)

(* Insert ERR *)		(* Repeat previous steps to create the log has to be transmitted on the network	*)
s1:=CONCAT('&ERR=',INT_TO_STRING(Level));
s1:=CONCAT(s1,';');
s1:=CONCAT(s1,INT_TO_STRING(Object));
s1:=CONCAT(s1,';');
s1:=CONCAT(s1,WORD_TO_STRING(Index));
s1:=CONCAT(s1,';');
s1:=CONCAT(s1,WORD_TO_STRING(Error));
s1:=CONCAT(s1,';');

ADDSTRING(ADR(Logger.TData), ADR(s1), Logger.TLen);		(* Add this part of the log to the previous one (the header)	*)
s1:=Message;
STR_NOSPACES(ADR(s1));									(* Check there are no blank spaces in the "Message"	*)
ADDSTRING(ADR(Logger.TData), ADR(s1), Logger.TLen);		(* Add error message to the rest of the log file	*)

(*---------------------------------------------------------------*)
	Logger_Send();
(*---------------------------------------------------------------*)
END_FUNCTION

(* POU TCP_Logger/LogTrig, ST *)
FUNCTION LogTrig : BOOL
VAR
	s1 : STRING(160);
	i  : BYTE;
END_VAR
(*---------------------------------------------------------------*)
	Logger_Head();
(*---------------------------------------------------------------*)

FOR i:=1 TO Plant_INV BY 1 DO
	INV[i].AddLogData(ModBus := MODB01);
END_FOR

FOR i:=1 TO Plant_STR BY 1 DO
	IF i<>7 THEN STR[i].AddLogData(ModBus := MODB01); END_IF
END_FOR

(*---------------------------------------------------------------*)
	Logger_Send();
(*---------------------------------------------------------------*)
END_FUNCTION

(* POU Utils Functions/MEMCLR, ST *)
FUNCTION MEMCLR:BOOL
VAR_INPUT
	pDestinationAddress:POINTER TO ARRAY[1..2] OF BYTE;
	BytesToClear:WORD;
END_VAR
VAR
END_VAR
WHILE (BytesToClear > 0) DO
	pDestinationAddress^[1]:=0;
	pDestinationAddress:=ADR(pDestinationAddress^[2]); (* increment destination *)
	BytesToClear:=BytesToClear -1; (* decrement number of bytes to copy *)
END_WHILE
END_FUNCTION

(* POU Plant_Objects/obj_MODBUS, ST *)
FUNCTION_BLOCK obj_MODBUS
(* === MODBUS PROTOCOL INTERFACE ===
   v1.1[19/06/15] - Added new VARS allocation and searching
*)
VAR CONSTANT
	VARS_Max	: BYTE := 32;
END_VAR
VAR_INPUT
	(* Settings *)
	ID			: BYTE;
	COM			: BYTE;
	BAUDRATE	: COM_BAUDRATE;
	RS485		: BOOL := FALSE;

	(* Interface *)
	MB_MASTER	: MODBUS_EXTENDED_MASTER;
	MB_Start	: BOOL;
	MB_Query	: typModbusExtendedQuery;
	MB_Resp		: typModbusResponse;
	MB_Lock		: BOOL;
	MB_Obj		: en_SYS_Objects;
	MB_ObjId	: BYTE;

	(* Variables management *)
	VARS_En		: BOOL := FALSE;
	VARS		: ARRAY [0..VARS_Max] OF typ_MODBUS_VAR;
	VARS_Check	: BOOL;
	VARS_Alarm	: BOOL;

	(* Variables allocation *)
	VAR_Pointer : POINTER TO ARRAY[0..99] OF WORD;
	VAR_Cfg		: POINTER TO typ_MODBUS_VAR;
END_VAR
VAR_OUTPUT
	(* Status *)
	Status_Log	: BYTE;
	Status_Vis	: DWORD;
END_VAR
VAR
	sta         : BYTE :=0;
	i			: BYTE;
	j			: BYTE;

	AlarmCOM	: FLT_EVENT;	(* Physical error relative to serial port -> COM	*)
	AlarmMDB	: FLT_EVENT;	(* ModBus error due to communication protocol error	*)

	VarTmr		: TON := (PT:=T#1s);
	VarSta		: BYTE; (* Status *)
	VarCnt		: BYTE; (* Scan counter *)
	VarRetry	: BYTE;
	VarAlarm	: BYTE; (* Last variable with errors *)
END_VAR
MB_MASTER(ENABLE:=TRUE,	ASCII_Mode:=FALSE, bCOM_PORT:=COM, cbCOM_BAUDRATE:=BAUDRATE, cpCOM_PARITY:=PARITY_NO,
		csCOM_STOPBITS:=STOPBITS_2,	cbsCOM_BYTESIZE:=BS_8, cfCOM_FLOW_CONTROL:=SEL(RS485,NO_FLOW_CONTROL,HALFDUPLEX),
		tTIME_OUT:=t#250ms,	StartFunction:=MB_Start, ExtQuery:=MB_Query, Response:=MB_Resp);

(* Process variable management *)
IF VARS_En THEN VARS_Process(); END_IF

(* Check status *)
AlarmCOM(IN:=(MB_MASTER.bInterfaceError<>0));
IF AlarmCOM.EVH THEN
	LogEv(SEL(MB_MASTER.bInterfaceError<>3,EL_Wrn,EL_Alarm),EO_MODBUS,ID,1,BYTE_TO_STRING(MB_MASTER.bInterfaceError));
END_IF
IF AlarmCOM.EVL THEN								(* Trigger a fall edge: MODBUS back working *)
	LogEv(EL_Log,EO_MODBUS,ID,2,'MODBUS_OK');
END_IF

(* If VARS not active check if a protocol error has occured (if VARS active this check is already done in "VARS_Process"	*)
IF NOT VARS_En THEN

	AlarmMDB(IN:=(MB_MASTER.MB_Error<>0));
(*	IF AlarmMDB.EVH THEN
		LogEv(EL_Wrn,EO_MODBUS,ID,2,INT_TO_STRING(MB_MASTER.MB_Error));
	END_IF
	IF AlarmMDB.EVL THEN								(* Trigger a fall edge: MODBUS back working *)
		LogEv(EL_Log,EO_MODBUS,ID,2,'MODBUS_OK');
	END_IF
*)
END_IF

(* Log/visu status *)
IF AlarmCOM.IN THEN Status_Log:=2; Status_Vis:=COLOR_RED;
ELSIF Vars_Alarm OR AlarmMDB.IN THEN Status_Log:=1; Status_Vis:=COLOR_YELLOW;
ELSE Status_Log:=0; Status_Vis:=COLOR_GREEN;
END_IF
END_FUNCTION_BLOCK
ACTION VAR_Search:
(* Search VAR with specific pointer if not found return first free VAR
	[Last VAR is not active... used as safe area...] 
*)
j:=VARS_Max;
FOR i := 0 TO VARS_Max-1 DO
	IF VARS[i].Variable=0 AND j>i THEN j:=i; END_IF
	IF VARS[i].Variable=VAR_Pointer THEN
		VAR_Cfg:=ADR(VARS[i]);
		RETURN;
	END_IF
END_FOR
VAR_Cfg:=ADR(VARS[j]);
END_ACTION
ACTION VARS_Process:
(* Update var timers *)
VarTmr(IN:=(NOT VarTmr.Q));
IF VarTmr.Q THEN
	FOR i := 0 TO VARS_Max DO
		IF VARS[i].Refresh_Cnt>0 THEN VARS[i].Refresh_Cnt:=VARS[i].Refresh_Cnt-1; END_IF
	END_FOR
	VARS_Check:=TRUE;
END_IF


(* Process status *)
CASE VarSta OF
	0: (* === Init *)
		VarCnt:=0;
		VarSta:=1;

	1: (* === Wait check signal *)
		IF VARS_Check THEN				(* Decremented "Refresh_Cnt" *)
			VARS_Check:=FALSE;
			VarCnt:=0;
			VarSta:=2;
		END_IF

	2: (* === Check loop *)
		IF NOT (MB_Lock OR MB_Start) THEN
			WHILE VarCnt<=(VARS_Max-1) AND VarSta=2 DO
				(* Check only active vars *)
				IF VARS[VarCnt].Variable<>0 THEN			(* "Variable" is a pointer to word, so if 0 no address *)
					(* Check var auto-refresh on timer checks *)
					IF VARS[VarCnt].Refresh_Time>0 AND VARS[VarCnt].Refresh_Cnt=0 THEN
						VARS[VarCnt].Refresh_Cnt:=VARS[VarCnt].Refresh_Time;
						VarSta:=3;
					END_IF
					(* Check refresh for change or request *)
					CASE VARS[VarCnt].FunCode OF
						5,6,15,16: (* Write functions *)
							IF VARS[VarCnt].Variable_Size=1 THEN
								IF VARS[VarCnt].Variable^[0]<>VARS[VarCnt].Variable_Mirror THEN
									VARS[VarCnt].Variable_Mirror:=VARS[VarCnt].Variable^[0];
									VarSta:=3;
								END_IF
							ELSE
								IF VARS[VarCnt].Variable_Mirror<>0 THEN
									VARS[VarCnt].Variable_Mirror:=0;
									VarSta:=3;
								END_IF
							END_IF
						1,2,3,4: (* Read functions *)
							IF VARS[VarCnt].Variable_Mirror<>0 THEN
								VARS[VarCnt].Variable_Mirror:=0;
								VarSta:=3;
							END_IF
					END_CASE
				END_IF
				(* Process query *)
				IF VarSta=3 THEN
					MB_Lock:=TRUE;
					MB_Query.SlaveAddress:=VARS[VarCnt].SlaveAddress;
					MB_Query.FunctionCode:=VARS[VarCnt].FunCode;
					CASE VARS[VarCnt].FunCode OF
						16#5,16#6,16#F,16#10:
							MB_Query.Read_Quantity:=0;
							MB_Query.Read_StartAddress:=0;
							MB_Query.Write_StartAddress:=VARS[VarCnt].FunAddress;
							MB_Query.Write_Quantity:=VARS[VarCnt].Variable_Size;
							IF VARS[VarCnt].Variable_Size=200 THEN
								COPY_32SWAP16(VARS[VarCnt].Variable, ADR(MB_Query.Write_Data[0]));
							ELSIF VARS[VarCnt].Variable_Size>1 THEN
								MEMCPY(VARS[VarCnt].Variable, ADR(MB_Query.Write_Data[0]), 2*VARS[VarCnt].Variable_Size);
							ELSE
								MB_Query.Write_Data[0]:=VARS[VarCnt].Variable^[0];
							END_IF
						16#1,16#2,16#3,16#4:
							MB_Query.Read_StartAddress:=VARS[VarCnt].FunAddress;
							IF VARS[VarCnt].Variable_Size=200 THEN MB_Query.Read_Quantity:=2; ELSE
							  MB_Query.Read_Quantity:=VARS[VarCnt].Variable_Size;
							END_IF
							MB_Query.Write_StartAddress:=0;
							MB_Query.Write_Quantity:=0;
					END_CASE
					VarRetry:=0;
					MB_Start:=TRUE;
				ELSE
					VarCnt:=VarCnt+1;
				END_IF
			END_WHILE
			(* Check loop completed -> no actions *)
			IF VarSta=2 THEN VarSta:=1; END_IF
		END_IF

	3: (* === Wait & process MB response *)
		IF NOT MB_Start THEN
			IF MB_MASTER.MB_Error=0 THEN
				CASE VARS[VarCnt].FunCode OF
					1,2,3,4:
						IF VARS[VarCnt].Variable_Size=200 THEN
							COPY_32SWAP16(ADR(MB_Resp.Data), VARS[VarCnt].Variable);
						ELSIF VARS[VarCnt].Variable_Size>1 THEN
							MEMCPY(ADR(MB_Resp.Data), VARS[VarCnt].Variable, 2*VARS[VarCnt].Variable_Size);
						ELSE
							VARS[VarCnt].Variable^[0]:=MB_Resp.Data[0];
						END_IF
				END_CASE
				MB_Lock:=FALSE;
				(* Signal error recovery *)
				IF VARS_Alarm=TRUE AND VarCnt=VarAlarm THEN
					LogEv(EL_Wrn,EO_MODBUS,ID,5,'');
					VARS_Alarm:=FALSE;
				END_IF
				(* Next var *)
				VarCnt:=VarCnt+1;
				VarSta:=2;
			ELSE
				IF VarRetry<3 THEN
					VarRetry:=VarRetry+1;
					MB_Start:=TRUE;
				ELSE
					MB_Lock:=FALSE;
					(* Signal error *)
					IF VARS_Alarm=FALSE THEN
						LogEv(EL_Wrn,EO_MODBUS,ID,3,INT_TO_STRING(MB_MASTER.MB_Error));
						VARS_Alarm:=TRUE;
						VarAlarm:=VarCnt-1;
					END_IF
					(* Next var *)
					VarCnt:=VarCnt+1;
					VarSta:=2;
				END_IF
			END_IF
		END_IF

ELSE
	VarSta:=0;
END_CASE
END_ACTION

(* POU Plant_Objects/obj_MODBUS_INV_SUNWAYTG, ST *)
FUNCTION_BLOCK obj_MODBUS_INV_SUNWAYTG
VAR CONSTANT
		(* States of normal modbus data reading *)
		WAIT_STATE		:	BYTE := 0;
		QUERY_MEAS_1	:	BYTE := 1;
		QUERY_STATUS	:	BYTE := 3;
		QUERY_INSULATION:	BYTE := 4;
		QUERY_MEAS_2	:	BYTE := 5;
		QUERY_MEAS_3	:	BYTE := 6;
		QUERY_MEAS_4	: 	BYTE := 7;
		QUERY_MEAS_5	:	BYTE := 8;
		QUERY_MEAS_6	:	BYTE := 9;
		QUERY_MEAS_7	:	BYTE := 10;
		QUERY_TIME		:	BYTE := 11;
		QUERY_FAULT_LIST:	BYTE := 12;
		READ_FAULT_LIST	:	BYTE := 13;
		QUERY_EVENT		:	BYTE := 14;
		READ_EVENT		:	BYTE := 15;
		END_READ		:	BYTE := 16;

		ERROR_STATE		:	BYTE := 100;

END_VAR
VAR_INPUT
		ID			:	BYTE;
		Address		:	BYTE;

		(* Refresh time *)
		RefreshTime	: 	TIME := T#1m;

		(* Read fault list *)
		FaultAddr	:	WORD;

		retryErrMax	:	BYTE := 15;		(* 15 minutes *)
END_VAR
VAR_IN_OUT
		ModBus		:	obj_MODBUS;
END_VAR
VAR_OUTPUT
		Status_Log	:	BYTE;
		Status_Vis	:	DWORD;
END_VAR
VAR

		InitOK		:	BOOL := FALSE;

		(* Inverter typical data structure	*)
		Data		:	typ_MODBUS_INV_SUNWAYTG;
		tempData	:	typ_MODBUS_INV_SUNWAYTG;
		FaultData	:	typ_MODBUS_INV_SUNWAYTG_His;
		EventData	:	ARRAY [1..16] OF typ_MODBUS_INV_SUNWAYTG_His;

		(* Modbus State machine variables	*)
		state		:	BYTE;
		last_state	:	BYTE;
		state_fault	:	BYTE;
		retry		:	BYTE;
		retryErr	:	BYTE;
		ReadTmr		:	TON := (PT:=t#5s);	(* Just to do a first ModBus read at the beginning *)
		fModbusAlr	:	BOOL;

		(* Event check variable	*)
		Alarm		:	FLT_EVENT;
		Event		:	FLT_EVENT;
		ModBusAlr	:	FLT_EVENT := (INITEV:=FALSE);
		InsulAlr	:	FLT_EVENT := (INITEV:=FALSE);
		OffsetEvt	:	FLT_EVENT;
		StatusOK	:	FLT_EVENT := (INITEV:=FALSE);
		AlarmCtr	:	BYTE;
		WarningCtr	:	BYTE;

		OldEvent	:	WORD;

		(* Memory variables	*)
		LastSuppTime:	DWORD;
		LastOpTime	:	DWORD;
		LastEvSuppTime	:	DWORD;

		(* AddLogData managing variables	*)
		Esup_adj	:	DWORD;

		(* General variables	*)
		counter		:	BYTE;
		s1			:	STRING;
		s2			:	STRING;

		fTimeout	:	BOOL;
END_VAR
IF NOT InitOK THEN
	ReadTmr.PT := WORD_TO_TIME(ID*2000);
	InitOK := TRUE;
END_IF

(* If "FaultAddr" equals 0 proceed with normal working, otherwise satisfy server request for fault list request	*)
IF FaultAddr=0 THEN

	(* State machine *)
	Stm();

	(* Check if an alarm has occured *)
	CheckAlarm();

	(* Verify if an energy counter reset has happened	*)
	CheckCtrReset();

ELSE
	(* Fault list state machine	*)
	StmFault();

END_IF

(* Set "Status_Log" according to actual object status	*)
IF AlarmCtr > 0 THEN
	Status_Log := 2;
	Status_Vis := COLOR_RED;
ELSIF WarningCtr > 0 THEN
	Status_Log := 1;
	Status_Vis := COLOR_YELLOW;
ELSE
	Status_Log := 0;

	StatusOK(IN:=(Status_Log=0));
	IF StatusOK.EVH THEN LogEv(EL_Log,EO_INV,ID,1,'Status_Ok'); END_IF

	Status_Vis := COLOR_GREEN;
END_IF
END_FUNCTION_BLOCK
ACTION AddLogData:
Logger.s1:=INSERT('&INV=',BYTE_TO_STRING(ID),4);
IF ID<10 THEN Logger.s1:=INSERT(Logger.s1,'0',4); END_IF

(* Create messagge to append to the log file in string format, containing the historical value for current alarm	*)
(* Inverter Status *)
Logger.s1:=CONCAT(Logger.s1,WORD_TO_STRING(Data.Status));				Logger.s1:=CONCAT(Logger.s1,';');

(* Energy measurements *)

(* Value adjustment according to acutal offset *)
Esup_adj := Data.Esup_ExtCtr1 + Offset[ID];

(* Energy measurements *)
Logger.s1:=CONCAT(Logger.s1,DWORD_TO_STRING(Esup_adj));					Logger.s1:=CONCAT(Logger.s1,';');
Logger.s1:=CONCAT(Logger.s1,DWORD_TO_STRING(Data.ExtCtr2));				Logger.s1:=CONCAT(Logger.s1,';');
Logger.s1:=CONCAT(Logger.s1,DWORD_TO_STRING(Data.Epv));					Logger.s1:=CONCAT(Logger.s1,';');

(* Mains measurements *)
Logger.s1:=CONCAT(Logger.s1,WORD_TO_STRING(Data.Vrms_rs));				Logger.s1:=CONCAT(Logger.s1,';');
Logger.s1:=CONCAT(Logger.s1,WORD_TO_STRING(Data.Vrms_st));				Logger.s1:=CONCAT(Logger.s1,';');
Logger.s1:=CONCAT(Logger.s1,WORD_TO_STRING(Data.Vrms_tr));				Logger.s1:=CONCAT(Logger.s1,';');
Logger.s1:=CONCAT(Logger.s1,WORD_TO_STRING(Data.Vrms_r));				Logger.s1:=CONCAT(Logger.s1,';');
Logger.s1:=CONCAT(Logger.s1,WORD_TO_STRING(Data.Vrms_s));				Logger.s1:=CONCAT(Logger.s1,';');
Logger.s1:=CONCAT(Logger.s1,WORD_TO_STRING(Data.Vrms_t));				Logger.s1:=CONCAT(Logger.s1,';');
Logger.s1:=CONCAT(Logger.s1,INT_TO_STRING(Data.Irms_r));				Logger.s1:=CONCAT(Logger.s1,';');
Logger.s1:=CONCAT(Logger.s1,INT_TO_STRING(Data.Irms_s));				Logger.s1:=CONCAT(Logger.s1,';');
Logger.s1:=CONCAT(Logger.s1,INT_TO_STRING(Data.Irms_t));				Logger.s1:=CONCAT(Logger.s1,';');
Logger.s1:=CONCAT(Logger.s1,WORD_TO_STRING(Data.Iimbalance));			Logger.s1:=CONCAT(Logger.s1,';');
Logger.s1:=CONCAT(Logger.s1,INT_TO_STRING(Data.P_r));					Logger.s1:=CONCAT(Logger.s1,';');
Logger.s1:=CONCAT(Logger.s1,INT_TO_STRING(Data.P_s));					Logger.s1:=CONCAT(Logger.s1,';');
Logger.s1:=CONCAT(Logger.s1,INT_TO_STRING(Data.P_t));					Logger.s1:=CONCAT(Logger.s1,';');
Logger.s1:=CONCAT(Logger.s1,INT_TO_STRING(Data.Pr_r));					Logger.s1:=CONCAT(Logger.s1,';');
Logger.s1:=CONCAT(Logger.s1,INT_TO_STRING(Data.Pr_s));					Logger.s1:=CONCAT(Logger.s1,';');
Logger.s1:=CONCAT(Logger.s1,INT_TO_STRING(Data.Pr_t));					Logger.s1:=CONCAT(Logger.s1,';');

(* PV measurements *)
Logger.s1:=CONCAT(Logger.s1,WORD_TO_STRING(Data.Vpv));					Logger.s1:=CONCAT(Logger.s1,';');
Logger.s1:=CONCAT(Logger.s1,WORD_TO_STRING(Data.Ipv));					Logger.s1:=CONCAT(Logger.s1,';');
Logger.s1:=CONCAT(Logger.s1,INT_TO_STRING(Data.Ppv));					Logger.s1:=CONCAT(Logger.s1,';');

(* Time (could be used as reference timing) *)
Logger.s1:=CONCAT(Logger.s1,DWORD_TO_STRING(Data.OpTime/300));			Logger.s1:=CONCAT(Logger.s1,';');
Logger.s1:=CONCAT(Logger.s1,DWORD_TO_STRING(Data.SuppTime/300));		Logger.s1:=CONCAT(Logger.s1,';');

(* Frequency and Temperature *)
Logger.s1:=CONCAT(Logger.s1,INT_TO_STRING(Data.f));						Logger.s1:=CONCAT(Logger.s1,';');
Logger.s1:=CONCAT(Logger.s1,INT_TO_STRING(Data.Tigbt));					Logger.s1:=CONCAT(Logger.s1,';');

(* Add log returned by the object	*)
Logger.s1:=CONCAT(Logger.s1,BYTE_TO_STRING(Status_Log));

(* Add the entire new string "s1" with the updated measurements to the one has to be transmitted	*)
ADDSTRING(ADR(Logger.TData), ADR(Logger.s1), Logger.TLen);
END_ACTION
ACTION AppendMeasure:
(* Used to add signifcant measurements when an alarm happens *)
s1 := WORD_TO_STRING(FaultData.AlarmID);					s1 := CONCAT(s1,';');
s1 := CONCAT(s1, DWORD_TO_STRING(FaultData.SuppTime/300));	s1 := CONCAT(s1,';');
s1 := CONCAT(s1, DWORD_TO_STRING(FaultData.OpTime/300));	s1 := CONCAT(s1,';');
s1 := CONCAT(s1, WORD_TO_STRING(FaultData.InvStatus));		s1 := CONCAT(s1,';');
s1 := CONCAT(s1, WORD_TO_STRING(FaultData.Vpv_ref));		s1 := CONCAT(s1,';');
s1 := CONCAT(s1, WORD_TO_STRING(FaultData.Vpv));			s1 := CONCAT(s1,';');
s1 := CONCAT(s1, WORD_TO_STRING(FaultData.Vmain));			s1 := CONCAT(s1,';');
s1 := CONCAT(s1, WORD_TO_STRING(FaultData.Status2));		s1 := CONCAT(s1,';');
s1 := CONCAT(s1, WORD_TO_STRING(FaultData.Status1));		s1 := CONCAT(s1,';');
s1 := CONCAT(s1, INT_TO_STRING(FaultData.Tboard));			s1 := CONCAT(s1,';');
s1 := CONCAT(s1, INT_TO_STRING(FaultData.Tigbt));			s1 := CONCAT(s1,';');
s1 := CONCAT(s1, INT_TO_STRING(FaultData.I_u));				s1 := CONCAT(s1,';');
s1 := CONCAT(s1, INT_TO_STRING(FaultData.I_v));				s1 := CONCAT(s1,';');
s1 := CONCAT(s1, INT_TO_STRING(FaultData.I_w));				s1 := CONCAT(s1,';');
s1 := CONCAT(s1, WORD_TO_STRING(FaultData.ClampStatus));	s1 := CONCAT(s1,';');
s1 := CONCAT(s1, WORD_TO_STRING(FaultData.DigOutput));		s1 := CONCAT(s1,';');
s1 := CONCAT(s1, WORD_TO_STRING(FaultData.IgbtFault));		s1 := CONCAT(s1,';');
s1 := CONCAT(s1, DWORD_TO_STRING(FaultData.Psupp));			s1 := CONCAT(s1,';');
s1 := CONCAT(s1, DWORD_TO_STRING(FaultData.Epv));
END_ACTION
ACTION CheckAlarm:
(*** Verify ModBus error	***)
ModbusAlr(IN:=fModbusAlr);

IF ModbusAlr.EVH THEN
	LogEv(EL_Alarm,EO_INV,ID,4,SEL(ModBus.MB_MASTER.MB_Error<>0,'0','1'));
	AlarmCtr := AlarmCtr + 1;
END_IF

IF ModbusAlr.EVL THEN
	LogEv(EL_Log,EO_INV,ID,8,'');
	AlarmCtr := SEL(AlarmCtr=0, AlarmCtr-1, 0);
END_IF

(*** General alarm	***)
Alarm(IN:=(Data.ActiveAlarm<>0), INITEV:=FALSE);

IF Alarm.EVH THEN
	IF LastSuppTime <> FaultData.SuppTime OR LastOpTime <> FaultData.OpTime THEN

		(* Log that an alarm has occured and add significant measurements	*)
		AppendMeasure();
		LogEv(EL_Alarm,EO_INV,ID,3,s1);

		AlarmCtr := AlarmCtr + 1;

		(* Keep trace of relative time at which last alarm occurs	*)
		LastSuppTime := FaultData.SuppTime;
		LastOpTime := FaultData.OpTime;
	END_IF
END_IF

(* A fall edge is detected: "ActiveAlarm" is now 0 *)
IF Alarm.EVL THEN AlarmCtr := SEL(AlarmCtr=0, AlarmCtr-1, 0);	END_IF

(*** Insulation alarm	***)
InsulAlr(IN:=(Data.Insulation=1));

IF InsulAlr.EVH THEN
		LogEv(EL_Alarm,EO_INV,ID,2,s1);
		AlarmCtr := AlarmCtr + 1;
END_IF

IF InsulAlr.EVL THEN AlarmCtr := SEL(AlarmCtr=0, AlarmCtr-1, 0); END_IF


(**** Check event ****)
Event(IN:=Data.Event=OldEvent);

IF Event.EVH THEN
	LogEv(EL_Evt,EO_INV,ID,7,WORD_TO_STRING(Data.Event));
	OldEvent := Data.Event;
END_IF
END_ACTION
ACTION CheckCtrReset:
(* Check if energy counter resetted - offset is passed as "data field" in the following way: Offset_High;Offset_Low
									  if no offset to update, value is 0 *)

IF InitOK AND (NOT fModbusAlr) AND (Sys.Status = 0 ) THEN

	OffsetEvt(IN:=(Old_Esup[ID] > Data.Esup_ExtCtr1));

	(* A counter reset has happened -->> Update offset and transmit it to the server	*)
	IF OffsetEvt.EVH THEN
		Offset[ID] := Offset[ID] + Old_Esup[ID];		(* Update offset high word *)
		LogEv(EL_Log,EO_INV,ID,6,DWORD_TO_STRING(Offset[ID]));
	END_IF

END_IF

(* updates previous counter memory for recognizing resets *)
Old_Esup[ID]:= Data.Esup_ExtCtr1;
END_ACTION
ACTION Stm:
CASE state OF

	WAIT_STATE:	(* Refresh time manager *)

		ReadTmr(IN:=NOT(ReadTmr.Q));
		IF ReadTmr.Q THEN

			ReadTmr.PT := RefreshTime;			(* Refresh timer range *)

			(* Reset state machine variables and counters *)
			retry	:= 0;
			counter := 0;
			last_state	:= WAIT_STATE;

			(* Start state machine	*)
			state := QUERY_MEAS_1;

		END_IF

	(****			 MEASUREMENTS			  ****)

	QUERY_MEAS_1:	(* External energy counters and energies *)
		IF NOT ModBus.MB_Start AND (NOT ModBus.MB_Lock OR retry>0) THEN
			ModBus.MB_Lock := TRUE;

			ModBus.MB_Obj := EO_INV;
			ModBus.MB_ObjId := ID;

			ModBus.MB_Query.SlaveAddress := Address;
			ModBus.MB_Query.FunctionCode := 16#3;
			ModBus.MB_Query.Read_StartAddress := 1663;
			ModBus.MB_Query.Read_Quantity := 6;
			ModBus.MB_Start := TRUE;

			state := QUERY_STATUS;
		END_IF

	QUERY_STATUS:	(* Status and Alarms *)

		IF NOT ModBus.MB_Start THEN
			IF ModBus.MB_MASTER.bInterfaceError<>0 OR ModBus.MB_MASTER.MB_Error<>0 THEN
				last_state := QUERY_MEAS_1;
				state := ERROR_STATE;
			ELSE

				tempData.Esup_ExtCtr1  	:= BUILD_16TO32_COPY(ModBus.MB_Resp.Data[0], ModBus.MB_Resp.Data[1]) ;
				tempData.ExtCtr2  		:= BUILD_16TO32_COPY(ModBus.MB_Resp.Data[2], ModBus.MB_Resp.Data[3]) ;
				tempData.Epv			:= BUILD_16TO32_COPY(ModBus.MB_Resp.Data[4], ModBus.MB_Resp.Data[5]) ;

				ModBus.MB_Query.SlaveAddress := Address;
				ModBus.MB_Query.FunctionCode := 16#3;
				ModBus.MB_Query.Read_StartAddress := 1739;
				ModBus.MB_Query.Read_Quantity := 2;
				ModBus.MB_Start := TRUE;

				state := QUERY_INSULATION;

			END_IF
		END_IF

	QUERY_INSULATION:	(* Insulation *)

		IF NOT ModBus.MB_Start THEN
			IF ModBus.MB_MASTER.bInterfaceError<>0 OR ModBus.MB_MASTER.MB_Error<>0 THEN
				last_state := QUERY_STATUS;
				state := ERROR_STATE;
			ELSE
				tempData.Status 	 := ModBus.MB_Resp.Data[0];
				tempData.ActiveAlarm := ModBus.MB_Resp.Data[1];

				ModBus.MB_Query.SlaveAddress := Address;
				ModBus.MB_Query.FunctionCode := 16#3;
				ModBus.MB_Query.Read_StartAddress := 1825;
				ModBus.MB_Query.Read_Quantity := 1;
				ModBus.MB_Start := TRUE;

				state := QUERY_MEAS_2;

			END_IF
		END_IF


	QUERY_MEAS_2:	(* Events *)
		IF NOT ModBus.MB_Start THEN
			IF ModBus.MB_MASTER.bInterfaceError<>0 OR ModBus.MB_MASTER.MB_Error<>0 THEN
				last_state := QUERY_INSULATION;
				state := ERROR_STATE;
			ELSE
				tempData.Insulation := ModBus.MB_Resp.Data[0];

				(* General measurements *)
				ModBus.MB_Query.SlaveAddress := Address;
				ModBus.MB_Query.FunctionCode := 16#3;
				ModBus.MB_Query.Read_StartAddress := 1650;
				ModBus.MB_Query.Read_Quantity := 13;
				ModBus.MB_Start := TRUE;

				state := QUERY_MEAS_3;
			END_IF
		END_IF

	QUERY_MEAS_3:	(* Cpu board and Igbt temperature *)

		IF NOT ModBus.MB_Start THEN
			IF ModBus.MB_MASTER.bInterfaceError<>0 OR ModBus.MB_MASTER.MB_Error<>0 THEN
				last_state := QUERY_MEAS_2;
				state := ERROR_STATE;
			ELSE
				tempData.Vpv_ref 	:= ModBus.MB_Resp.Data[0];
				tempData.f 			:= WORD_TO_INT(ModBus.MB_Resp.Data[1]);
				tempData.pf 		:= ModBus.MB_Resp.Data[2];
				tempData.P 			:= WORD_TO_INT(ModBus.MB_Resp.Data[3]);
				tempData.Pr 		:= WORD_TO_INT(ModBus.MB_Resp.Data[4]);
				tempData.Pa 		:= WORD_TO_INT(ModBus.MB_Resp.Data[5]);
				tempData.Vinv 		:= ModBus.MB_Resp.Data[6];
				tempData.Vmain 		:= ModBus.MB_Resp.Data[7];
				tempData.Iinv 		:= ModBus.MB_Resp.Data[8];
				tempData.Imain 		:= ModBus.MB_Resp.Data[9];
				tempData.Vpv 		:= ModBus.MB_Resp.Data[10];
				tempData.Ipv 		:= ModBus.MB_Resp.Data[11];
				tempData.Ppv 		:= WORD_TO_INT(ModBus.MB_Resp.Data[12]);

				ModBus.MB_Query.SlaveAddress := Address;
				ModBus.MB_Query.FunctionCode := 16#3;
				ModBus.MB_Query.Read_StartAddress := 1712;
				ModBus.MB_Query.Read_Quantity := 3;
				ModBus.MB_Start := TRUE;

				state := QUERY_MEAS_4;
			END_IF
		END_IF

	QUERY_MEAS_4:	(* Digital inputs *)

		IF NOT ModBus.MB_Start THEN
			IF ModBus.MB_MASTER.bInterfaceError<>0 OR ModBus.MB_MASTER.MB_Error<>0 THEN
				last_state := QUERY_MEAS_3;
				state := ERROR_STATE;
			ELSE
				tempData.Tboard := WORD_TO_INT(ModBus.MB_Resp.Data[0]);
				tempData.Tigbt 	:= WORD_TO_INT(ModBus.MB_Resp.Data[2]);

				ModBus.MB_Query.SlaveAddress := Address;
				ModBus.MB_Query.FunctionCode := 16#3;
				ModBus.MB_Query.Read_StartAddress := 1682;
				ModBus.MB_Query.Read_Quantity := 1;
				ModBus.MB_Start := TRUE;

				state := QUERY_MEAS_5;
			END_IF
		END_IF

	QUERY_MEAS_5:	(* Mains measurements *)

		IF NOT ModBus.MB_Start THEN
			IF ModBus.MB_MASTER.bInterfaceError<>0 OR ModBus.MB_MASTER.MB_Error<>0 THEN
				last_state := QUERY_MEAS_4;
				state := ERROR_STATE;
			ELSE
				tempData.ClampStatus := ModBus.MB_Resp.Data[0];

				ModBus.MB_Query.SlaveAddress := Address;
				ModBus.MB_Query.FunctionCode := 16#3;
				ModBus.MB_Query.Read_StartAddress := 1687;
				ModBus.MB_Query.Read_Quantity := 13;
				ModBus.MB_Start := TRUE;

				state := QUERY_MEAS_6;
			END_IF
		END_IF

	QUERY_MEAS_6:	(* Mains measurements *)

		IF NOT ModBus.MB_Start THEN
			IF ModBus.MB_MASTER.bInterfaceError<>0 OR ModBus.MB_MASTER.MB_Error<>0 THEN
				last_state := QUERY_MEAS_5;
				state := ERROR_STATE;
			ELSE
				tempData.Vrms_rs 		:= ModBus.MB_Resp.Data[0];
				tempData.Vrms_st 		:= ModBus.MB_Resp.Data[1];
				tempData.Vrms_tr 		:= ModBus.MB_Resp.Data[2];
				tempData.Irms_r 		:= WORD_TO_INT(ModBus.MB_Resp.Data[3]);
				tempData.Irms_s 		:= WORD_TO_INT(ModBus.MB_Resp.Data[4]);
				tempData.Irms_t 		:= WORD_TO_INT(ModBus.MB_Resp.Data[5]);
				tempData.PLLStatus 		:= ModBus.MB_Resp.Data[6];
				tempData.MainStatus2 	:= ModBus.MB_Resp.Data[7];
				tempData.MainStatus1 	:= ModBus.MB_Resp.Data[8];
				tempData.Iinv_rms_r 	:= WORD_TO_INT(ModBus.MB_Resp.Data[9]);
				tempData.Iinv_rms_s 	:= WORD_TO_INT(ModBus.MB_Resp.Data[10]);
				tempData.Iinv_rms_t 	:= WORD_TO_INT(ModBus.MB_Resp.Data[11]);
				tempData.Iimbalance		:= ModBus.MB_Resp.Data[12];

				ModBus.MB_Query.SlaveAddress := Address;
				ModBus.MB_Query.FunctionCode := 16#3;
				ModBus.MB_Query.Read_StartAddress := 1715;
				ModBus.MB_Query.Read_Quantity := 3;
				ModBus.MB_Start := TRUE;

				state := QUERY_MEAS_7;
			END_IF
		END_IF

	QUERY_MEAS_7:	(* Mains measurements *)

		IF NOT ModBus.MB_Start THEN
			IF ModBus.MB_MASTER.bInterfaceError<>0 OR ModBus.MB_MASTER.MB_Error<>0 THEN
				last_state := QUERY_MEAS_6;
				state := ERROR_STATE;
			ELSE
				tempData.Vrms_r	:= ModBus.MB_Resp.Data[0];
				tempData.Vrms_s := ModBus.MB_Resp.Data[1];
				tempData.Vrms_t := ModBus.MB_Resp.Data[2];

				ModBus.MB_Query.SlaveAddress := Address;
				ModBus.MB_Query.FunctionCode := 16#3;
				ModBus.MB_Query.Read_StartAddress := 1721;
				ModBus.MB_Query.Read_Quantity := 6;
				ModBus.MB_Start := TRUE;

				state := QUERY_TIME;
			END_IF
		END_IF

	QUERY_TIME:	(* Supply and operation time *)

		IF NOT ModBus.MB_Start THEN
			IF ModBus.MB_MASTER.bInterfaceError<>0 OR ModBus.MB_MASTER.MB_Error<>0 THEN
				last_state := QUERY_MEAS_7;
				state := ERROR_STATE;
			ELSE
				tempData.P_r	:= WORD_TO_INT(ModBus.MB_Resp.Data[0]);
				tempData.P_s 	:= WORD_TO_INT(ModBus.MB_Resp.Data[1]);
				tempData.P_t 	:= WORD_TO_INT(ModBus.MB_Resp.Data[2]);
				tempData.Pr_r	:= WORD_TO_INT(ModBus.MB_Resp.Data[3]);
				tempData.Pr_s 	:= WORD_TO_INT(ModBus.MB_Resp.Data[4]);
				tempData.Pr_t 	:= WORD_TO_INT(ModBus.MB_Resp.Data[5]);

				ModBus.MB_Query.SlaveAddress := Address;
				ModBus.MB_Query.FunctionCode := 16#3;
				ModBus.MB_Query.Read_StartAddress := 1702;
				ModBus.MB_Query.Read_Quantity := 4;
				ModBus.MB_Start := TRUE;

				state := QUERY_FAULT_LIST;
			END_IF
		END_IF

	QUERY_FAULT_LIST:	(* If an alarm has occured, read last fault list *)

		IF NOT ModBus.MB_Start THEN
			IF ModBus.MB_MASTER.bInterfaceError<>0 OR ModBus.MB_MASTER.MB_Error<>0 THEN
				last_state := QUERY_TIME;
				state := ERROR_STATE;
			ELSE
				tempData.OpTime := BUILD_16TO32_COPY(ModBus.MB_Resp.Data[0],ModBus.MB_Resp.Data[1]);
				tempData.SuppTime := BUILD_16TO32_COPY(ModBus.MB_Resp.Data[2],ModBus.MB_Resp.Data[3]);

				IF Data.ActiveAlarm <> 0 THEN

					ModBus.MB_Query.SlaveAddress := Address;
					ModBus.MB_Query.FunctionCode := 16#3;
					ModBus.MB_Query.Read_StartAddress := 7712;
					ModBus.MB_Query.Read_Quantity := 23;
					ModBus.MB_Start := TRUE;

					state := READ_FAULT_LIST;

				ELSE
					state := QUERY_EVENT;
				END_IF
			END_IF
		END_IF

	READ_FAULT_LIST:

		IF NOT ModBus.MB_Start THEN
			IF ModBus.MB_MASTER.bInterfaceError<>0 OR ModBus.MB_MASTER.MB_Error<>0 THEN
				last_state := QUERY_FAULT_LIST;
				state := ERROR_STATE;
			ELSE
				FaultData.AlarmID 		:= ModBus.MB_Resp.Data[0];
				FaultData.SuppTime 		:= BUILD_16TO32_COPY(ModBus.MB_Resp.Data[1],ModBus.MB_Resp.Data[2]);
				FaultData.OpTime 		:= BUILD_16TO32_COPY(ModBus.MB_Resp.Data[3],ModBus.MB_Resp.Data[4]);
				FaultData.InvStatus 	:= ModBus.MB_Resp.Data[5];
				FaultData.Vpv_ref 		:= ModBus.MB_Resp.Data[6];
				FaultData.Vpv 			:= ModBus.MB_Resp.Data[7];
				FaultData.Vmain 		:= ModBus.MB_Resp.Data[8];
				FaultData.Status2 		:= ModBus.MB_Resp.Data[9];
				FaultData.Status1 		:= ModBus.MB_Resp.Data[10];
				FaultData.Tboard 		:= ModBus.MB_Resp.Data[11];
				FaultData.Tigbt 		:= ModBus.MB_Resp.Data[12];
				FaultData.I_u 			:= ModBus.MB_Resp.Data[13];
				FaultData.I_v 			:= ModBus.MB_Resp.Data[14];
				FaultData.I_w 			:= ModBus.MB_Resp.Data[15];
				FaultData.ClampStatus 	:= ModBus.MB_Resp.Data[16];
				FaultData.DigOutput 	:= ModBus.MB_Resp.Data[17];
				FaultData.IgbtFault 	:= ModBus.MB_Resp.Data[18];
				FaultData.Psupp			:= BUILD_16TO32_COPY(ModBus.MB_Resp.Data[19],ModBus.MB_Resp.Data[20]);
				FaultData.Epv 			:= BUILD_16TO32_COPY(ModBus.MB_Resp.Data[21],ModBus.MB_Resp.Data[22]);

				state := QUERY_EVENT;

			END_IF
		END_IF

	QUERY_EVENT:

		IF NOT ModBus.MB_Start THEN
			IF ModBus.MB_MASTER.bInterfaceError<>0 OR ModBus.MB_MASTER.MB_Error<>0 THEN
				last_state := READ_FAULT_LIST;
				state := ERROR_STATE;
			ELSE

				(* Read all 16 events data	*)
				ModBus.MB_Query.SlaveAddress := Address;
				ModBus.MB_Query.FunctionCode := 16#3;
				ModBus.MB_Query.Read_StartAddress := 5044;
				ModBus.MB_Query.Read_Quantity := 1;
				ModBus.MB_Start := TRUE;

				state := READ_EVENT;

			END_IF
		END_IF

	READ_EVENT:

		IF NOT ModBus.MB_Start THEN
			IF ModBus.MB_MASTER.bInterfaceError<>0 OR (ModBus.MB_MASTER.MB_Error<>0 AND ModBus.MB_MASTER.MB_Error<MB_TIME_OUT) THEN
				last_state := QUERY_EVENT;
				state := ERROR_STATE;
			ELSE
				tempData.Event	:= ModBus.MB_Resp.Data[0];

				(* Copy temporary read data *)
				MEMCPY(ADR(tempData), ADR(Data), SIZEOF(Data));

				fModbusAlr := FALSE;
				retryErr := 0;
				ModBus.MB_Lock := FALSE;
				state := WAIT_STATE;

				(*** TEST ***)
				fTimeout := FALSE;
			END_IF
		END_IF


	ERROR_STATE:	(* Error state *)

		IF retry < 3 THEN
			retry := retry+1;
			state := last_state;

		ELSE
			ModBus.MB_Lock := FALSE;

			(* Verify if slave is dead *)
			IF retryErr < retryErrMaX THEN
				retryErr := retryErr + 1;
			ELSE
				fModbusAlr := TRUE;
			END_IF

			(* Back to wait state *)
			state := WAIT_STATE;

			(*** TEST ***)
			fTimeout := TRUE;
		END_IF

		IF ModBus.MB_MASTER.MB_Error=MB_TIME_OUT THEN
			state := state;
		END_IF
ELSE
	state := WAIT_STATE;
END_CASE
END_ACTION
ACTION StmFault:
(* State machine *)
CASE state_fault OF

	WAIT_STATE:
		IF NOT (ModBus.MB_Lock OR ModBus.MB_Start) THEN
			ModBus.MB_Lock := TRUE;
			counter := 0;
			retry 	:= 0;
			last_state  := WAIT_STATE;
			state_fault := QUERY_FAULT_LIST;
		ELSE
			last_state  := WAIT_STATE;
			state_fault := ERROR_STATE;
		END_IF

	QUERY_FAULT_LIST:

			ModBus.MB_Query.SlaveAddress := Address;
			ModBus.MB_Query.FunctionCode := 16#3;
			ModBus.MB_Query.Read_Quantity := 24;
			ModBus.MB_Query.Read_StartAddress := FaultAddr;
			ModBus.MB_Start := TRUE;

			state_fault := READ_FAULT_LIST;

	READ_FAULT_LIST:
		IF NOT ModBus.MB_Start THEN
			IF ModBus.MB_MASTER.bInterfaceError<>0 OR ModBus.MB_MASTER.MB_Error<>0 THEN

				last_state := QUERY_FAULT_LIST;
				state := ERROR_STATE;

			ELSE

